MoveL RelTool (p1,64.500000,13.500000,11.989951,\Rx:=0.000000,\Ry:=0.000000),vel1,zoneval,Extruder\WObj:=Workobject_1;
MoveL RelTool (p1,65.000000,13.500000,11.512795,\Rx:=0.000000,\Ry:=0.000000),vel1,zoneval,Extruder\WObj:=Workobject_1;
MoveL RelTool (p1,65.500000,13.500000,11.007442,\Rx:=0.000000,\Ry:=0.000000),vel1,zoneval,Extruder\WObj:=Workobject_1;
MoveL RelTool (p1,66.000000,13.500000,10.423269,\Rx:=0.000000,\Ry:=0.000000),vel1,zoneval,Extruder\WObj:=Workobject_1;
MoveL RelTool (p1,66.500000,13.500000,9.763981,\Rx:=0.000000,\Ry:=0.000000),vel1,zoneval,Extruder\WObj:=Workobject_1;
MoveL RelTool (p1,67.000000,13.500000,9.225973,\Rx:=0.000000,\Ry:=0.000000),vel1,zoneval,Extruder\WObj:=Workobject_1;
MoveL RelTool (p1,67.500000,13.500000,8.874086,\Rx:=0.000000,\Ry:=0.000000),vel1,zoneval,Extruder\WObj:=Workobject_1;
MoveL RelTool (p1,68.000000,13.500000,8.652682,\Rx:=0.000000,\Ry:=0.000000),vel1,zoneval,Extruder\WObj:=Workobject_1;
MoveL RelTool (p1,68.500000,13.500000,8.535785,\Rx:=0.000000,\Ry:=0.000000),vel1,zoneval,Extruder\WObj:=Workobject_1;
MoveL RelTool (p1,69.000000,13.500000,8.500000,\Rx:=0.000000,\Ry:=0.000000),vel1,zoneval,Extruder\WObj:=Workobject_1;
MoveL RelTool (p1,69.500000,13.500000,8.500000,\Rx:=0.000000,\Ry:=0.000000),vel1,zoneval,Extruder\WObj:=Workobject_1;
MoveL RelTool (p1,70.000000,13.500000,8.500000,\Rx:=0.000000,\Ry:=0.000000),vel1,zoneval,Extruder\WObj:=Workobject_1;
MoveL RelTool (p1,70.500000,13.500000,8.500000,\Rx:=0.000000,\Ry:=0.000000),vel1,zoneval,Extruder\WObj:=Workobject_1;
MoveL RelTool (p1,71.000000,13.500000,8.500000,\Rx:=0.000000,\Ry:=0.000000),vel1,zoneval,Extruder\WObj:=Workobject_1;
MoveL RelTool (p1,71.500000,13.500000,8.500000,\Rx:=0.000000,\Ry:=0.000000),vel1,zoneval,Extruder\WObj:=Workobject_1;
MoveL RelTool (p1,72.000000,13.500000,8.500000,\Rx:=0.000000,\Ry:=0.000000),vel1,zoneval,Extruder\WObj:=Workobject_1;
MoveL RelTool (p1,72.500000,13.500000,8.500000,\Rx:=0.000000,\Ry:=0.000000),vel1,zoneval,Extruder\WObj:=Workobject_1;
MoveL RelTool (p1,73.000000,13.500000,8.500000,\Rx:=0.000000,\Ry:=0.000000),vel1,zoneval,Extruder\WObj:=Workobject_1;
MoveL RelTool (p1,73.500000,13.500000,8.500000,\Rx:=0.000000,\Ry:=0.000000),vel1,zoneval,Extruder\WObj:=Workobject_1;
MoveL RelTool (p1,74.000000,13.500000,8.500000,\Rx:=0.000000,\Ry:=0.000000),vel1,zoneval,Extruder\WObj:=Workobject_1;
MoveL RelTool (p1,74.500000,13.500000,8.500000,\Rx:=0.000000,\Ry:=0.000000),vel1,zoneval,Extruder\WObj:=Workobject_1;
MoveL RelTool (p1,75.000000,13.500000,8.500000,\Rx:=0.000000,\Ry:=0.000000),vel1,zoneval,Extruder\WObj:=Workobject_1;
MoveL RelTool (p1,75.500000,13.500000,8.500000,\Rx:=0.000000,\Ry:=0.000000),vel1,zoneval,Extruder\WObj:=Workobject_1;
MoveL RelTool (p1,76.000000,13.500000,8.500000,\Rx:=0.000000,\Ry:=0.000000),vel1,zoneval,Extruder\WObj:=Workobject_1;
MoveL RelTool (p1,76.500000,13.500000,8.500000,\Rx:=0.000000,\Ry:=0.000000),vel1,zoneval,Extruder\WObj:=Workobject_1;
MoveL RelTool (p1,77.000000,13.500000,8.500000,\Rx:=0.000000,\Ry:=0.000000),vel1,zoneval,Extruder\WObj:=Workobject_1;
MoveL RelTool (p1,77.500000,13.500000,8.500000,\Rx:=0.000000,\Ry:=0.000000),vel1,zoneval,Extruder\WObj:=Workobject_1;
MoveL RelTool (p1,78.000000,13.500000,8.500000,\Rx:=0.000000,\Ry:=0.000000),vel1,zoneval,Extruder\WObj:=Workobject_1;
MoveL RelTool (p1,78.500000,13.500000,8.500000,\Rx:=0.000000,\Ry:=0.000000),vel1,zoneval,Extruder\WObj:=Workobject_1;
MoveL RelTool (p1,79.000000,13.500000,8.500000,\Rx:=0.000000,\Ry:=0.000000),vel1,zoneval,Extruder\WObj:=Workobject_1;
MoveL RelTool (p1,79.500000,13.500000,8.500000,\Rx:=0.000000,\Ry:=0.000000),vel1,zoneval,Extruder\WObj:=Workobject_1;
MoveL RelTool (p1,80.000000,13.500000,8.500000,\Rx:=0.000000,\Ry:=0.000000),vel1,zoneval,Extruder\WObj:=Workobject_1;
MoveL RelTool (p1,80.500000,13.500000,8.500000,\Rx:=0.000000,\Ry:=0.000000),vel1,zoneval,Extruder\WObj:=Workobject_1;
MoveL RelTool (p1,81.000000,13.500000,8.500000,\Rx:=0.000000,\Ry:=0.000000),vel1,zoneval,Extruder\WObj:=Workobject_1;
MoveL RelTool (p1,81.500000,13.500000,8.500000,\Rx:=0.000000,\Ry:=0.000000),vel1,zoneval,Extruder\WObj:=Workobject_1;
MoveL RelTool (p1,82.000000,13.500000,8.500000,\Rx:=0.000000,\Ry:=0.000000),vel1,zoneval,Extruder\WObj:=Workobject_1;
MoveL RelTool (p1,82.000000,14.000000,8.500000,\Rx:=0.000000,\Ry:=0.000000),vel1,zoneval,Extruder\WObj:=Workobject_1;
MoveL RelTool (p1,81.500000,14.000000,8.500000,\Rx:=0.000000,\Ry:=0.000000),vel1,zoneval,Extruder\WObj:=Workobject_1;
MoveL RelTool (p1,81.000000,14.000000,8.500000,\Rx:=0.000000,\Ry:=0.000000),vel1,zoneval,Extruder\WObj:=Workobject_1;
MoveL RelTool (p1,80.500000,14.000000,8.500000,\Rx:=0.000000,\Ry:=0.000000),vel1,zoneval,Extruder\WObj:=Workobject_1;
MoveL RelTool (p1,80.000000,14.000000,8.500000,\Rx:=0.000000,\Ry:=0.000000),vel1,zoneval,Extruder\WObj:=Workobject_1;
MoveL RelTool (p1,79.500000,14.000000,8.500000,\Rx:=0.000000,\Ry:=0.000000),vel1,zoneval,Extruder\WObj:=Workobject_1;
MoveL RelTool (p1,79.000000,14.000000,8.500000,\Rx:=0.000000,\Ry:=0.000000),vel1,zoneval,Extruder\WObj:=Workobject_1;
MoveL RelTool (p1,78.500000,14.000000,8.500000,\Rx:=0.000000,\Ry:=0.000000),vel1,zoneval,Extruder\WObj:=Workobject_1;
MoveL RelTool (p1,78.000000,14.000000,8.500000,\Rx:=0.000000,\Ry:=0.000000),vel1,zoneval,Extruder\WObj:=Workobject_1;
MoveL RelTool (p1,77.500000,14.000000,8.500000,\Rx:=0.000000,\Ry:=0.000000),vel1,zoneval,Extruder\WObj:=Workobject_1;
MoveL RelTool (p1,77.000000,14.000000,8.500000,\Rx:=0.000000,\Ry:=0.000000),vel1,zoneval,Extruder\WObj:=Workobject_1;
MoveL RelTool (p1,76.500000,14.000000,8.500000,\Rx:=0.000000,\Ry:=0.000000),vel1,zoneval,Extruder\WObj:=Workobject_1;
MoveL RelTool (p1,76.000000,14.000000,8.500000,\Rx:=0.000000,\Ry:=0.000000),vel1,zoneval,Extruder\WObj:=Workobject_1;
MoveL RelTool (p1,75.500000,14.000000,8.500000,\Rx:=0.000000,\Ry:=0.000000),vel1,zoneval,Extruder\WObj:=Workobject_1;
MoveL RelTool (p1,75.000000,14.000000,8.500000,\Rx:=0.000000,\Ry:=0.000000),vel1,zoneval,Extruder\WObj:=Workobject_1;
MoveL RelTool (p1,74.500000,14.000000,8.500000,\Rx:=0.000000,\Ry:=0.000000),vel1,zoneval,Extruder\WObj:=Workobject_1;
MoveL RelTool (p1,74.000000,14.000000,8.500000,\Rx:=0.000000,\Ry:=0.000000),vel1,zoneval,Extruder\WObj:=Workobject_1;
MoveL RelTool (p1,73.500000,14.000000,8.500000,\Rx:=0.000000,\Ry:=0.000000),vel1,zoneval,Extruder\WObj:=Workobject_1;
MoveL RelTool (p1,73.000000,14.000000,8.500000,\Rx:=0.000000,\Ry:=0.000000),vel1,zoneval,Extruder\WObj:=Workobject_1;
MoveL RelTool (p1,72.500000,14.000000,8.500000,\Rx:=0.000000,\Ry:=0.000000),vel1,zoneval,Extruder\WObj:=Workobject_1;
MoveL RelTool (p1,72.000000,14.000000,8.500000,\Rx:=0.000000,\Ry:=0.000000),vel1,zoneval,Extruder\WObj:=Workobject_1;
MoveL RelTool (p1,71.500000,14.000000,8.500000,\Rx:=0.000000,\Ry:=0.000000),vel1,zoneval,Extruder\WObj:=Workobject_1;
MoveL RelTool (p1,71.000000,14.000000,8.500000,\Rx:=0.000000,\Ry:=0.000000),vel1,zoneval,Extruder\WObj:=Workobject_1;
MoveL RelTool (p1,70.500000,14.000000,8.500000,\Rx:=0.000000,\Ry:=0.000000),vel1,zoneval,Extruder\WObj:=Workobject_1;
MoveL RelTool (p1,70.000000,14.000000,8.500000,\Rx:=0.000000,\Ry:=0.000000),vel1,zoneval,Extruder\WObj:=Workobject_1;
MoveL RelTool (p1,69.500000,14.000000,8.500000,\Rx:=0.000000,\Ry:=0.000000),vel1,zoneval,Extruder\WObj:=Workobject_1;
MoveL RelTool (p1,69.000000,14.000000,8.500000,\Rx:=0.000000,\Ry:=0.000000),vel1,zoneval,Extruder\WObj:=Workobject_1;
MoveL RelTool (p1,68.500000,14.000000,8.535785,\Rx:=0.000000,\Ry:=0.000000),vel1,zoneval,Extruder\WObj:=Workobject_1;
MoveL RelTool (p1,68.000000,14.000000,8.652682,\Rx:=0.000000,\Ry:=0.000000),vel1,zoneval,Extruder\WObj:=Workobject_1;
MoveL RelTool (p1,67.500000,14.000000,8.874086,\Rx:=0.000000,\Ry:=0.000000),vel1,zoneval,Extruder\WObj:=Workobject_1;
MoveL RelTool (p1,67.000000,14.000000,9.225973,\Rx:=0.000000,\Ry:=0.000000),vel1,zoneval,Extruder\WObj:=Workobject_1;
MoveL RelTool (p1,66.500000,14.000000,9.763981,\Rx:=0.000000,\Ry:=0.000000),vel1,zoneval,Extruder\WObj:=Workobject_1;
MoveL RelTool (p1,66.000000,14.000000,10.424782,\Rx:=0.000000,\Ry:=0.000000),vel1,zoneval,Extruder\WObj:=Workobject_1;
MoveL RelTool (p1,65.500000,14.000000,11.007081,\Rx:=0.000000,\Ry:=0.000000),vel1,zoneval,Extruder\WObj:=Workobject_1;
MoveL RelTool (p1,65.000000,14.000000,11.513962,\Rx:=0.000000,\Ry:=0.000000),vel1,zoneval,Extruder\WObj:=Workobject_1;
MoveL RelTool (p1,64.500000,14.000000,11.989543,\Rx:=0.000000,\Ry:=0.000000),vel1,zoneval,Extruder\WObj:=Workobject_1;
MoveL RelTool (p1,64.000000,14.000000,12.421528,\Rx:=0.000000,\Ry:=0.000000),vel1,zoneval,Extruder\WObj:=Workobject_1;
MoveL RelTool (p1,63.500000,14.000000,12.805855,\Rx:=0.000000,\Ry:=0.000000),vel1,zoneval,Extruder\WObj:=Workobject_1;
MoveL RelTool (p1,63.000000,14.000000,13.179500,\Rx:=0.000000,\Ry:=0.000000),vel1,zoneval,Extruder\WObj:=Workobject_1;
MoveL RelTool (p1,62.500000,14.000000,13.514872,\Rx:=0.000000,\Ry:=0.000000),vel1,zoneval,Extruder\WObj:=Workobject_1;
MoveL RelTool (p1,62.000000,14.000000,13.838447,\Rx:=0.000000,\Ry:=0.000000),vel1,zoneval,Extruder\WObj:=Workobject_1;
MoveL RelTool (p1,61.500000,14.000000,14.134422,\Rx:=0.000000,\Ry:=0.000000),vel1,zoneval,Extruder\WObj:=Workobject_1;
MoveL RelTool (p1,61.000000,14.000000,14.418567,\Rx:=0.000000,\Ry:=0.000000),vel1,zoneval,Extruder\WObj:=Workobject_1;
MoveL RelTool (p1,60.500000,14.000000,14.677184,\Rx:=0.000000,\Ry:=0.000000),vel1,zoneval,Extruder\WObj:=Workobject_1;
MoveL RelTool (p1,60.000000,14.000000,14.938229,\Rx:=0.000000,\Ry:=0.000000),vel1,zoneval,Extruder\WObj:=Workobject_1;
MoveL RelTool (p1,59.500000,14.000000,15.174609,\Rx:=0.000000,\Ry:=0.000000),vel1,zoneval,Extruder\WObj:=Workobject_1;
MoveL RelTool (p1,59.000000,14.000000,15.404406,\Rx:=0.000000,\Ry:=0.000000),vel1,zoneval,Extruder\WObj:=Workobject_1;
MoveL RelTool (p1,58.500000,14.000000,15.614404,\Rx:=0.000000,\Ry:=0.000000),vel1,zoneval,Extruder\WObj:=Workobject_1;
MoveL RelTool (p1,58.000000,14.000000,15.816030,\Rx:=0.000000,\Ry:=0.000000),vel1,zoneval,Extruder\WObj:=Workobject_1;
MoveL RelTool (p1,57.500000,14.000000,16.017656,\Rx:=0.000000,\Ry:=0.000000),vel1,zoneval,Extruder\WObj:=Workobject_1;
MoveL RelTool (p1,57.000000,14.000000,16.197291,\Rx:=0.000000,\Ry:=0.000000),vel1,zoneval,Extruder\WObj:=Workobject_1;
MoveL RelTool (p1,56.500000,14.000000,16.373201,\Rx:=0.000000,\Ry:=0.000000),vel1,zoneval,Extruder\WObj:=Workobject_1;
MoveL RelTool (p1,56.000000,14.000000,16.541775,\Rx:=0.000000,\Ry:=0.000000),vel1,zoneval,Extruder\WObj:=Workobject_1;
MoveL RelTool (p1,55.500000,14.000000,16.695933,\Rx:=0.000000,\Ry:=0.000000),vel1,zoneval,Extruder\WObj:=Workobject_1;
MoveL RelTool (p1,55.000000,14.000000,16.847549,\Rx:=0.000000,\Ry:=0.000000),vel1,zoneval,Extruder\WObj:=Workobject_1;
MoveL RelTool (p1,54.500000,14.000000,16.992424,\Rx:=0.000000,\Ry:=0.000000),vel1,zoneval,Extruder\WObj:=Workobject_1;
MoveL RelTool (p1,54.000000,14.000000,17.116147,\Rx:=0.000000,\Ry:=0.000000),vel1,zoneval,Extruder\WObj:=Workobject_1;
MoveL RelTool (p1,53.500000,14.000000,17.244747,\Rx:=0.000000,\Ry:=0.000000),vel1,zoneval,Extruder\WObj:=Workobject_1;
MoveL RelTool (p1,53.000000,14.000000,17.373347,\Rx:=0.000000,\Ry:=0.000000),vel1,zoneval,Extruder\WObj:=Workobject_1;
MoveL RelTool (p1,52.500000,14.000000,17.484402,\Rx:=0.000000,\Ry:=0.000000),vel1,zoneval,Extruder\WObj:=Workobject_1;
MoveL RelTool (p1,52.000000,14.000000,17.591158,\Rx:=0.000000,\Ry:=0.000000),vel1,zoneval,Extruder\WObj:=Workobject_1;
MoveL RelTool (p1,51.500000,14.000000,17.695333,\Rx:=0.000000,\Ry:=0.000000),vel1,zoneval,Extruder\WObj:=Workobject_1;
MoveL RelTool (p1,51.000000,14.000000,17.779951,\Rx:=0.000000,\Ry:=0.000000),vel1,zoneval,Extruder\WObj:=Workobject_1;
MoveL RelTool (p1,50.500000,14.000000,17.865927,\Rx:=0.000000,\Ry:=0.000000),vel1,zoneval,Extruder\WObj:=Workobject_1;
MoveL RelTool (p1,50.000000,14.000000,17.951904,\Rx:=0.000000,\Ry:=0.000000),vel1,zoneval,Extruder\WObj:=Workobject_1;
MoveL RelTool (p1,49.500000,14.000000,18.029069,\Rx:=0.000000,\Ry:=0.000000),vel1,zoneval,Extruder\WObj:=Workobject_1;
MoveL RelTool (p1,49.000000,14.000000,18.095126,\Rx:=0.000000,\Ry:=0.000000),vel1,zoneval,Extruder\WObj:=Workobject_1;
MoveL RelTool (p1,48.500000,14.000000,18.161183,\Rx:=0.000000,\Ry:=0.000000),vel1,zoneval,Extruder\WObj:=Workobject_1;
MoveL RelTool (p1,48.000000,14.000000,18.218591,\Rx:=0.000000,\Ry:=0.000000),vel1,zoneval,Extruder\WObj:=Workobject_1;
MoveL RelTool (p1,47.500000,14.000000,18.266605,\Rx:=0.000000,\Ry:=0.000000),vel1,zoneval,Extruder\WObj:=Workobject_1;
MoveL RelTool (p1,47.000000,14.000000,18.313237,\Rx:=0.000000,\Ry:=0.000000),vel1,zoneval,Extruder\WObj:=Workobject_1;
MoveL RelTool (p1,46.500000,14.000000,18.359868,\Rx:=0.000000,\Ry:=0.000000),vel1,zoneval,Extruder\WObj:=Workobject_1;
MoveL RelTool (p1,46.000000,14.000000,18.393525,\Rx:=0.000000,\Ry:=0.000000),vel1,zoneval,Extruder\WObj:=Workobject_1;
MoveL RelTool (p1,45.500000,14.000000,18.421069,\Rx:=0.000000,\Ry:=0.000000),vel1,zoneval,Extruder\WObj:=Workobject_1;
MoveL RelTool (p1,45.000000,14.000000,18.448613,\Rx:=0.000000,\Ry:=0.000000),vel1,zoneval,Extruder\WObj:=Workobject_1;
MoveL RelTool (p1,44.500000,14.000000,18.469450,\Rx:=0.000000,\Ry:=0.000000),vel1,zoneval,Extruder\WObj:=Workobject_1;
MoveL RelTool (p1,44.000000,14.000000,18.480446,\Rx:=0.000000,\Ry:=0.000000),vel1,zoneval,Extruder\WObj:=Workobject_1;
MoveL RelTool (p1,43.500000,14.000000,18.488975,\Rx:=0.000000,\Ry:=0.000000),vel1,zoneval,Extruder\WObj:=Workobject_1;
MoveL RelTool (p1,43.000000,14.000000,18.497504,\Rx:=0.000000,\Ry:=0.000000),vel1,zoneval,Extruder\WObj:=Workobject_1;
MoveL RelTool (p1,42.500000,14.000000,18.493713,\Rx:=0.000000,\Ry:=0.000000),vel1,zoneval,Extruder\WObj:=Workobject_1;
MoveL RelTool (p1,42.000000,14.000000,18.483301,\Rx:=0.000000,\Ry:=0.000000),vel1,zoneval,Extruder\WObj:=Workobject_1;
MoveL RelTool (p1,41.500000,14.000000,18.472889,\Rx:=0.000000,\Ry:=0.000000),vel1,zoneval,Extruder\WObj:=Workobject_1;
MoveL RelTool (p1,41.000000,14.000000,18.457063,\Rx:=0.000000,\Ry:=0.000000),vel1,zoneval,Extruder\WObj:=Workobject_1;
MoveL RelTool (p1,40.500000,14.000000,18.431185,\Rx:=0.000000,\Ry:=0.000000),vel1,zoneval,Extruder\WObj:=Workobject_1;
MoveL RelTool (p1,40.000000,14.000000,18.401735,\Rx:=0.000000,\Ry:=0.000000),vel1,zoneval,Extruder\WObj:=Workobject_1;
MoveL RelTool (p1,39.500000,14.000000,18.372284,\Rx:=0.000000,\Ry:=0.000000),vel1,zoneval,Extruder\WObj:=Workobject_1;
MoveL RelTool (p1,39.000000,14.000000,18.328181,\Rx:=0.000000,\Ry:=0.000000),vel1,zoneval,Extruder\WObj:=Workobject_1;
MoveL RelTool (p1,38.500000,14.000000,18.278194,\Rx:=0.000000,\Ry:=0.000000),vel1,zoneval,Extruder\WObj:=Workobject_1;
MoveL RelTool (p1,38.000000,14.000000,18.229591,\Rx:=0.000000,\Ry:=0.000000),vel1,zoneval,Extruder\WObj:=Workobject_1;
MoveL RelTool (p1,37.500000,14.000000,18.180988,\Rx:=0.000000,\Ry:=0.000000),vel1,zoneval,Extruder\WObj:=Workobject_1;
MoveL RelTool (p1,37.000000,14.000000,18.118155,\Rx:=0.000000,\Ry:=0.000000),vel1,zoneval,Extruder\WObj:=Workobject_1;
MoveL RelTool (p1,36.500000,14.000000,18.049890,\Rx:=0.000000,\Ry:=0.000000),vel1,zoneval,Extruder\WObj:=Workobject_1;
MoveL RelTool (p1,36.000000,14.000000,17.981627,\Rx:=0.000000,\Ry:=0.000000),vel1,zoneval,Extruder\WObj:=Workobject_1;
MoveL RelTool (p1,35.500000,14.000000,17.897001,\Rx:=0.000000,\Ry:=0.000000),vel1,zoneval,Extruder\WObj:=Workobject_1;
MoveL RelTool (p1,35.000000,14.000000,17.808427,\Rx:=0.000000,\Ry:=0.000000),vel1,zoneval,Extruder\WObj:=Workobject_1;
MoveL RelTool (p1,34.500000,14.000000,17.719854,\Rx:=0.000000,\Ry:=0.000000),vel1,zoneval,Extruder\WObj:=Workobject_1;
MoveL RelTool (p1,34.000000,14.000000,17.630421,\Rx:=0.000000,\Ry:=0.000000),vel1,zoneval,Extruder\WObj:=Workobject_1;
MoveL RelTool (p1,33.500000,14.000000,17.520494,\Rx:=0.000000,\Ry:=0.000000),vel1,zoneval,Extruder\WObj:=Workobject_1;
MoveL RelTool (p1,33.000000,14.000000,17.410567,\Rx:=0.000000,\Ry:=0.000000),vel1,zoneval,Extruder\WObj:=Workobject_1;
MoveL RelTool (p1,32.500000,14.000000,17.295270,\Rx:=0.000000,\Ry:=0.000000),vel1,zoneval,Extruder\WObj:=Workobject_1;
MoveL RelTool (p1,32.000000,14.000000,17.166180,\Rx:=0.000000,\Ry:=0.000000),vel1,zoneval,Extruder\WObj:=Workobject_1;
MoveL RelTool (p1,31.500000,14.000000,17.033775,\Rx:=0.000000,\Ry:=0.000000),vel1,zoneval,Extruder\WObj:=Workobject_1;
MoveL RelTool (p1,31.000000,14.000000,16.901371,\Rx:=0.000000,\Ry:=0.000000),vel1,zoneval,Extruder\WObj:=Workobject_1;
MoveL RelTool (p1,30.500000,14.000000,16.748138,\Rx:=0.000000,\Ry:=0.000000),vel1,zoneval,Extruder\WObj:=Workobject_1;
MoveL RelTool (p1,30.000000,14.000000,16.592069,\Rx:=0.000000,\Ry:=0.000000),vel1,zoneval,Extruder\WObj:=Workobject_1;
MoveL RelTool (p1,29.500000,14.000000,16.432055,\Rx:=0.000000,\Ry:=0.000000),vel1,zoneval,Extruder\WObj:=Workobject_1;
MoveL RelTool (p1,29.000000,14.000000,16.256775,\Rx:=0.000000,\Ry:=0.000000),vel1,zoneval,Extruder\WObj:=Workobject_1;
MoveL RelTool (p1,28.500000,14.000000,16.075776,\Rx:=0.000000,\Ry:=0.000000),vel1,zoneval,Extruder\WObj:=Workobject_1;
MoveL RelTool (p1,28.000000,14.000000,15.889441,\Rx:=0.000000,\Ry:=0.000000),vel1,zoneval,Extruder\WObj:=Workobject_1;
MoveL RelTool (p1,27.500000,14.000000,15.681605,\Rx:=0.000000,\Ry:=0.000000),vel1,zoneval,Extruder\WObj:=Workobject_1;
MoveL RelTool (p1,27.000000,14.000000,15.473770,\Rx:=0.000000,\Ry:=0.000000),vel1,zoneval,Extruder\WObj:=Workobject_1;
MoveL RelTool (p1,26.500000,14.000000,15.254742,\Rx:=0.000000,\Ry:=0.000000),vel1,zoneval,Extruder\WObj:=Workobject_1;
MoveL RelTool (p1,26.000000,14.000000,15.016990,\Rx:=0.000000,\Ry:=0.000000),vel1,zoneval,Extruder\WObj:=Workobject_1;
MoveL RelTool (p1,25.500000,14.000000,14.773856,\Rx:=0.000000,\Ry:=0.000000),vel1,zoneval,Extruder\WObj:=Workobject_1;
MoveL RelTool (p1,25.000000,14.000000,14.503734,\Rx:=0.000000,\Ry:=0.000000),vel1,zoneval,Extruder\WObj:=Workobject_1;
MoveL RelTool (p1,24.500000,14.000000,14.232533,\Rx:=0.000000,\Ry:=0.000000),vel1,zoneval,Extruder\WObj:=Workobject_1;
MoveL RelTool (p1,24.000000,14.000000,13.937132,\Rx:=0.000000,\Ry:=0.000000),vel1,zoneval,Extruder\WObj:=Workobject_1;
MoveL RelTool (p1,23.500000,14.000000,13.628434,\Rx:=0.000000,\Ry:=0.000000),vel1,zoneval,Extruder\WObj:=Workobject_1;
MoveL RelTool (p1,23.000000,14.000000,13.289112,\Rx:=0.000000,\Ry:=0.000000),vel1,zoneval,Extruder\WObj:=Workobject_1;
MoveL RelTool (p1,22.500000,14.000000,12.938180,\Rx:=0.000000,\Ry:=0.000000),vel1,zoneval,Extruder\WObj:=Workobject_1;
MoveL RelTool (p1,22.000000,14.000000,12.548317,\Rx:=0.000000,\Ry:=0.000000),vel1,zoneval,Extruder\WObj:=Workobject_1;
MoveL RelTool (p1,21.500000,14.000000,12.139462,\Rx:=0.000000,\Ry:=0.000000),vel1,zoneval,Extruder\WObj:=Workobject_1;
MoveL RelTool (p1,21.000000,14.000000,11.683424,\Rx:=0.000000,\Ry:=0.000000),vel1,zoneval,Extruder\WObj:=Workobject_1;
MoveL RelTool (p1,20.500000,14.000000,11.178595,\Rx:=0.000000,\Ry:=0.000000),vel1,zoneval,Extruder\WObj:=Workobject_1;
MoveL RelTool (p1,20.000000,14.000000,10.625965,\Rx:=0.000000,\Ry:=0.000000),vel1,zoneval,Extruder\WObj:=Workobject_1;
MoveL RelTool (p1,19.500000,14.000000,9.992651,\Rx:=0.000000,\Ry:=0.000000),vel1,zoneval,Extruder\WObj:=Workobject_1;
MoveL RelTool (p1,19.000000,14.000000,9.374813,\Rx:=0.000000,\Ry:=0.000000),vel1,zoneval,Extruder\WObj:=Workobject_1;
MoveL RelTool (p1,18.500000,14.000000,8.980296,\Rx:=0.000000,\Ry:=0.000000),vel1,zoneval,Extruder\WObj:=Workobject_1;
MoveL RelTool (p1,18.000000,14.000000,8.722633,\Rx:=0.000000,\Ry:=0.000000),vel1,zoneval,Extruder\WObj:=Workobject_1;
MoveL RelTool (p1,17.500000,14.000000,8.570628,\Rx:=0.000000,\Ry:=0.000000),vel1,zoneval,Extruder\WObj:=Workobject_1;
MoveL RelTool (p1,17.000000,14.000000,8.508911,\Rx:=0.000000,\Ry:=0.000000),vel1,zoneval,Extruder\WObj:=Workobject_1;
MoveL RelTool (p1,16.500000,14.000000,8.500000,\Rx:=0.000000,\Ry:=0.000000),vel1,zoneval,Extruder\WObj:=Workobject_1;
MoveL RelTool (p1,16.000000,14.000000,8.500000,\Rx:=0.000000,\Ry:=0.000000),vel1,zoneval,Extruder\WObj:=Workobject_1;
MoveL RelTool (p1,15.500000,14.000000,8.500000,\Rx:=0.000000,\Ry:=0.000000),vel1,zoneval,Extruder\WObj:=Workobject_1;
MoveL RelTool (p1,15.000000,14.000000,8.500000,\Rx:=0.000000,\Ry:=0.000000),vel1,zoneval,Extruder\WObj:=Workobject_1;
MoveL RelTool (p1,14.500000,14.000000,8.500000,\Rx:=0.000000,\Ry:=0.000000),vel1,zoneval,Extruder\WObj:=Workobject_1;
MoveL RelTool (p1,14.000000,14.000000,8.500000,\Rx:=0.000000,\Ry:=0.000000),vel1,zoneval,Extruder\WObj:=Workobject_1;
MoveL RelTool (p1,13.500000,14.000000,8.500000,\Rx:=0.000000,\Ry:=0.000000),vel1,zoneval,Extruder\WObj:=Workobject_1;
MoveL RelTool (p1,13.000000,14.000000,8.500000,\Rx:=0.000000,\Ry:=0.000000),vel1,zoneval,Extruder\WObj:=Workobject_1;
MoveL RelTool (p1,12.500000,14.000000,8.500000,\Rx:=0.000000,\Ry:=0.000000),vel1,zoneval,Extruder\WObj:=Workobject_1;
MoveL RelTool (p1,12.000000,14.000000,8.500000,\Rx:=0.000000,\Ry:=0.000000),vel1,zoneval,Extruder\WObj:=Workobject_1;
MoveL RelTool (p1,11.500000,14.000000,8.500000,\Rx:=0.000000,\Ry:=0.000000),vel1,zoneval,Extruder\WObj:=Workobject_1;
MoveL RelTool (p1,11.000000,14.000000,8.500000,\Rx:=0.000000,\Ry:=0.000000),vel1,zoneval,Extruder\WObj:=Workobject_1;
MoveL RelTool (p1,10.500000,14.000000,8.500000,\Rx:=0.000000,\Ry:=0.000000),vel1,zoneval,Extruder\WObj:=Workobject_1;
MoveL RelTool (p1,10.000000,14.000000,8.500000,\Rx:=0.000000,\Ry:=0.000000),vel1,zoneval,Extruder\WObj:=Workobject_1;
MoveL RelTool (p1,9.500000,14.000000,8.500000,\Rx:=0.000000,\Ry:=0.000000),vel1,zoneval,Extruder\WObj:=Workobject_1;
MoveL RelTool (p1,9.000000,14.000000,8.500000,\Rx:=0.000000,\Ry:=0.000000),vel1,zoneval,Extruder\WObj:=Workobject_1;
MoveL RelTool (p1,8.500000,14.000000,8.500000,\Rx:=0.000000,\Ry:=0.000000),vel1,zoneval,Extruder\WObj:=Workobject_1;
MoveL RelTool (p1,8.000000,14.000000,8.500000,\Rx:=0.000000,\Ry:=0.000000),vel1,zoneval,Extruder\WObj:=Workobject_1;
MoveL RelTool (p1,7.500000,14.000000,8.500000,\Rx:=0.000000,\Ry:=0.000000),vel1,zoneval,Extruder\WObj:=Workobject_1;
MoveL RelTool (p1,7.000000,14.000000,8.500000,\Rx:=0.000000,\Ry:=0.000000),vel1,zoneval,Extruder\WObj:=Workobject_1;
MoveL RelTool (p1,6.500000,14.000000,8.500000,\Rx:=0.000000,\Ry:=0.000000),vel1,zoneval,Extruder\WObj:=Workobject_1;
MoveL RelTool (p1,6.000000,14.000000,8.500000,\Rx:=0.000000,\Ry:=0.000000),vel1,zoneval,Extruder\WObj:=Workobject_1;
MoveL RelTool (p1,5.500000,14.000000,8.500000,\Rx:=0.000000,\Ry:=0.000000),vel1,zoneval,Extruder\WObj:=Workobject_1;
MoveL RelTool (p1,5.000000,14.000000,8.500000,\Rx:=0.000000,\Ry:=0.000000),vel1,zoneval,Extruder\WObj:=Workobject_1;
MoveL RelTool (p1,4.500000,14.000000,8.500000,\Rx:=0.000000,\Ry:=0.000000),vel1,zoneval,Extruder\WObj:=Workobject_1;
MoveL RelTool (p1,4.000000,14.000000,8.500000,\Rx:=0.000000,\Ry:=0.000000),vel1,zoneval,Extruder\WObj:=Workobject_1;
MoveL RelTool (p1,3.500000,14.000000,8.500000,\Rx:=0.000000,\Ry:=0.000000),vel1,zoneval,Extruder\WObj:=Workobject_1;
MoveL RelTool (p1,3.500000,14.500000,8.500000,\Rx:=0.000000,\Ry:=0.000000),vel1,zoneval,Extruder\WObj:=Workobject_1;
MoveL RelTool (p1,4.000000,14.500000,8.500000,\Rx:=0.000000,\Ry:=0.000000),vel1,zoneval,Extruder\WObj:=Workobject_1;
MoveL RelTool (p1,4.500000,14.500000,8.500000,\Rx:=0.000000,\Ry:=0.000000),vel1,zoneval,Extruder\WObj:=Workobject_1;
MoveL RelTool (p1,5.000000,14.500000,8.500000,\Rx:=0.000000,\Ry:=0.000000),vel1,zoneval,Extruder\WObj:=Workobject_1;
MoveL RelTool (p1,5.500000,14.500000,8.500000,\Rx:=0.000000,\Ry:=0.000000),vel1,zoneval,Extruder\WObj:=Workobject_1;
MoveL RelTool (p1,6.000000,14.500000,8.500000,\Rx:=0.000000,\Ry:=0.000000),vel1,zoneval,Extruder\WObj:=Workobject_1;
MoveL RelTool (p1,6.500000,14.500000,8.500000,\Rx:=0.000000,\Ry:=0.000000),vel1,zoneval,Extruder\WObj:=Workobject_1;
MoveL RelTool (p1,7.000000,14.500000,8.500000,\Rx:=0.000000,\Ry:=0.000000),vel1,zoneval,Extruder\WObj:=Workobject_1;
MoveL RelTool (p1,7.500000,14.500000,8.500000,\Rx:=0.000000,\Ry:=0.000000),vel1,zoneval,Extruder\WObj:=Workobject_1;
MoveL RelTool (p1,8.000000,14.500000,8.500000,\Rx:=0.000000,\Ry:=0.000000),vel1,zoneval,Extruder\WObj:=Workobject_1;
MoveL RelTool (p1,8.500000,14.500000,8.500000,\Rx:=0.000000,\Ry:=0.000000),vel1,zoneval,Extruder\WObj:=Workobject_1;
MoveL RelTool (p1,9.000000,14.500000,8.500000,\Rx:=0.000000,\Ry:=0.000000),vel1,zoneval,Extruder\WObj:=Workobject_1;
MoveL RelTool (p1,9.500000,14.500000,8.500000,\Rx:=0.000000,\Ry:=0.000000),vel1,zoneval,Extruder\WObj:=Workobject_1;
MoveL RelTool (p1,10.000000,14.500000,8.500000,\Rx:=0.000000,\Ry:=0.000000),vel1,zoneval,Extruder\WObj:=Workobject_1;
MoveL RelTool (p1,10.500000,14.500000,8.500000,\Rx:=0.000000,\Ry:=0.000000),vel1,zoneval,Extruder\WObj:=Workobject_1;
MoveL RelTool (p1,11.000000,14.500000,8.500000,\Rx:=0.000000,\Ry:=0.000000),vel1,zoneval,Extruder\WObj:=Workobject_1;
MoveL RelTool (p1,11.500000,14.500000,8.500000,\Rx:=0.000000,\Ry:=0.000000),vel1,zoneval,Extruder\WObj:=Workobject_1;
MoveL RelTool (p1,12.000000,14.500000,8.500000,\Rx:=0.000000,\Ry:=0.000000),vel1,zoneval,Extruder\WObj:=Workobject_1;
MoveL RelTool (p1,12.500000,14.500000,8.500000,\Rx:=0.000000,\Ry:=0.000000),vel1,zoneval,Extruder\WObj:=Workobject_1;
MoveL RelTool (p1,13.000000,14.500000,8.500000,\Rx:=0.000000,\Ry:=0.000000),vel1,zoneval,Extruder\WObj:=Workobject_1;
MoveL RelTool (p1,13.500000,14.500000,8.500000,\Rx:=0.000000,\Ry:=0.000000),vel1,zoneval,Extruder\WObj:=Workobject_1;
MoveL RelTool (p1,14.000000,14.500000,8.500000,\Rx:=0.000000,\Ry:=0.000000),vel1,zoneval,Extruder\WObj:=Workobject_1;
MoveL RelTool (p1,14.500000,14.500000,8.500000,\Rx:=0.000000,\Ry:=0.000000),vel1,zoneval,Extruder\WObj:=Workobject_1;
MoveL RelTool (p1,15.000000,14.500000,8.500000,\Rx:=0.000000,\Ry:=0.000000),vel1,zoneval,Extruder\WObj:=Workobject_1;
MoveL RelTool (p1,15.500000,14.500000,8.500000,\Rx:=0.000000,\Ry:=0.000000),vel1,zoneval,Extruder\WObj:=Workobject_1;
MoveL RelTool (p1,16.000000,14.500000,8.500000,\Rx:=0.000000,\Ry:=0.000000),vel1,zoneval,Extruder\WObj:=Workobject_1;
MoveL RelTool (p1,16.500000,14.500000,8.500000,\Rx:=0.000000,\Ry:=0.000000),vel1,zoneval,Extruder\WObj:=Workobject_1;
MoveL RelTool (p1,17.000000,14.500000,8.508911,\Rx:=0.000000,\Ry:=0.000000),vel1,zoneval,Extruder\WObj:=Workobject_1;
MoveL RelTool (p1,17.500000,14.500000,8.570628,\Rx:=0.000000,\Ry:=0.000000),vel1,zoneval,Extruder\WObj:=Workobject_1;
MoveL RelTool (p1,18.000000,14.500000,8.722633,\Rx:=0.000000,\Ry:=0.000000),vel1,zoneval,Extruder\WObj:=Workobject_1;
MoveL RelTool (p1,18.500000,14.500000,8.980296,\Rx:=0.000000,\Ry:=0.000000),vel1,zoneval,Extruder\WObj:=Workobject_1;
MoveL RelTool (p1,19.000000,14.500000,9.374813,\Rx:=0.000000,\Ry:=0.000000),vel1,zoneval,Extruder\WObj:=Workobject_1;
MoveL RelTool (p1,19.500000,14.500000,9.992651,\Rx:=0.000000,\Ry:=0.000000),vel1,zoneval,Extruder\WObj:=Workobject_1;
MoveL RelTool (p1,20.000000,14.500000,10.625441,\Rx:=0.000000,\Ry:=0.000000),vel1,zoneval,Extruder\WObj:=Workobject_1;
MoveL RelTool (p1,20.500000,14.500000,11.179034,\Rx:=0.000000,\Ry:=0.000000),vel1,zoneval,Extruder\WObj:=Workobject_1;
MoveL RelTool (p1,21.000000,14.500000,11.683147,\Rx:=0.000000,\Ry:=0.000000),vel1,zoneval,Extruder\WObj:=Workobject_1;
MoveL RelTool (p1,21.500000,14.500000,12.140800,\Rx:=0.000000,\Ry:=0.000000),vel1,zoneval,Extruder\WObj:=Workobject_1;
MoveL RelTool (p1,22.000000,14.500000,12.548217,\Rx:=0.000000,\Ry:=0.000000),vel1,zoneval,Extruder\WObj:=Workobject_1;
MoveL RelTool (p1,22.500000,14.500000,12.938300,\Rx:=0.000000,\Ry:=0.000000),vel1,zoneval,Extruder\WObj:=Workobject_1;
MoveL RelTool (p1,23.000000,14.500000,13.289231,\Rx:=0.000000,\Ry:=0.000000),vel1,zoneval,Extruder\WObj:=Workobject_1;
MoveL RelTool (p1,23.500000,14.500000,13.628094,\Rx:=0.000000,\Ry:=0.000000),vel1,zoneval,Extruder\WObj:=Workobject_1;
MoveL RelTool (p1,24.000000,14.500000,13.936792,\Rx:=0.000000,\Ry:=0.000000),vel1,zoneval,Extruder\WObj:=Workobject_1;
MoveL RelTool (p1,24.500000,14.500000,14.233179,\Rx:=0.000000,\Ry:=0.000000),vel1,zoneval,Extruder\WObj:=Workobject_1;
MoveL RelTool (p1,25.000000,14.500000,14.504380,\Rx:=0.000000,\Ry:=0.000000),vel1,zoneval,Extruder\WObj:=Workobject_1;
MoveL RelTool (p1,25.500000,14.500000,14.774776,\Rx:=0.000000,\Ry:=0.000000),vel1,zoneval,Extruder\WObj:=Workobject_1;
MoveL RelTool (p1,26.000000,14.500000,15.016632,\Rx:=0.000000,\Ry:=0.000000),vel1,zoneval,Extruder\WObj:=Workobject_1;
MoveL RelTool (p1,26.500000,14.500000,15.254383,\Rx:=0.000000,\Ry:=0.000000),vel1,zoneval,Extruder\WObj:=Workobject_1;
MoveL RelTool (p1,27.000000,14.500000,15.474110,\Rx:=0.000000,\Ry:=0.000000),vel1,zoneval,Extruder\WObj:=Workobject_1;
MoveL RelTool (p1,27.500000,14.500000,15.681946,\Rx:=0.000000,\Ry:=0.000000),vel1,zoneval,Extruder\WObj:=Workobject_1;
MoveL RelTool (p1,28.000000,14.500000,15.889782,\Rx:=0.000000,\Ry:=0.000000),vel1,zoneval,Extruder\WObj:=Workobject_1;
MoveL RelTool (p1,28.500000,14.500000,16.075557,\Rx:=0.000000,\Ry:=0.000000),vel1,zoneval,Extruder\WObj:=Workobject_1;
MoveL RelTool (p1,29.000000,14.500000,16.256557,\Rx:=0.000000,\Ry:=0.000000),vel1,zoneval,Extruder\WObj:=Workobject_1;
MoveL RelTool (p1,29.500000,14.500000,16.433092,\Rx:=0.000000,\Ry:=0.000000),vel1,zoneval,Extruder\WObj:=Workobject_1;
MoveL RelTool (p1,30.000000,14.500000,16.591990,\Rx:=0.000000,\Ry:=0.000000),vel1,zoneval,Extruder\WObj:=Workobject_1;
MoveL RelTool (p1,30.500000,14.500000,16.748059,\Rx:=0.000000,\Ry:=0.000000),vel1,zoneval,Extruder\WObj:=Workobject_1;
MoveL RelTool (p1,31.000000,14.500000,16.901521,\Rx:=0.000000,\Ry:=0.000000),vel1,zoneval,Extruder\WObj:=Workobject_1;
MoveL RelTool (p1,31.500000,14.500000,17.033926,\Rx:=0.000000,\Ry:=0.000000),vel1,zoneval,Extruder\WObj:=Workobject_1;
MoveL RelTool (p1,32.000000,14.500000,17.166330,\Rx:=0.000000,\Ry:=0.000000),vel1,zoneval,Extruder\WObj:=Workobject_1;
MoveL RelTool (p1,32.500000,14.500000,17.296270,\Rx:=0.000000,\Ry:=0.000000),vel1,zoneval,Extruder\WObj:=Workobject_1;
MoveL RelTool (p1,33.000000,14.500000,17.410275,\Rx:=0.000000,\Ry:=0.000000),vel1,zoneval,Extruder\WObj:=Workobject_1;
MoveL RelTool (p1,33.500000,14.500000,17.520202,\Rx:=0.000000,\Ry:=0.000000),vel1,zoneval,Extruder\WObj:=Workobject_1;
MoveL RelTool (p1,34.000000,14.500000,17.630129,\Rx:=0.000000,\Ry:=0.000000),vel1,zoneval,Extruder\WObj:=Workobject_1;
MoveL RelTool (p1,34.500000,14.500000,17.720622,\Rx:=0.000000,\Ry:=0.000000),vel1,zoneval,Extruder\WObj:=Workobject_1;
MoveL RelTool (p1,35.000000,14.500000,17.809195,\Rx:=0.000000,\Ry:=0.000000),vel1,zoneval,Extruder\WObj:=Workobject_1;
MoveL RelTool (p1,35.500000,14.500000,17.897769,\Rx:=0.000000,\Ry:=0.000000),vel1,zoneval,Extruder\WObj:=Workobject_1;
MoveL RelTool (p1,36.000000,14.500000,17.981309,\Rx:=0.000000,\Ry:=0.000000),vel1,zoneval,Extruder\WObj:=Workobject_1;
MoveL RelTool (p1,36.500000,14.500000,18.049573,\Rx:=0.000000,\Ry:=0.000000),vel1,zoneval,Extruder\WObj:=Workobject_1;
MoveL RelTool (p1,37.000000,14.500000,18.117838,\Rx:=0.000000,\Ry:=0.000000),vel1,zoneval,Extruder\WObj:=Workobject_1;
MoveL RelTool (p1,37.500000,14.500000,18.182228,\Rx:=0.000000,\Ry:=0.000000),vel1,zoneval,Extruder\WObj:=Workobject_1;
MoveL RelTool (p1,38.000000,14.500000,18.230831,\Rx:=0.000000,\Ry:=0.000000),vel1,zoneval,Extruder\WObj:=Workobject_1;
MoveL RelTool (p1,38.500000,14.500000,18.279434,\Rx:=0.000000,\Ry:=0.000000),vel1,zoneval,Extruder\WObj:=Workobject_1;
MoveL RelTool (p1,39.000000,14.500000,18.328464,\Rx:=0.000000,\Ry:=0.000000),vel1,zoneval,Extruder\WObj:=Workobject_1;
MoveL RelTool (p1,39.500000,14.500000,18.372133,\Rx:=0.000000,\Ry:=0.000000),vel1,zoneval,Extruder\WObj:=Workobject_1;
MoveL RelTool (p1,40.000000,14.500000,18.401583,\Rx:=0.000000,\Ry:=0.000000),vel1,zoneval,Extruder\WObj:=Workobject_1;
MoveL RelTool (p1,40.500000,14.500000,18.431033,\Rx:=0.000000,\Ry:=0.000000),vel1,zoneval,Extruder\WObj:=Workobject_1;
MoveL RelTool (p1,41.000000,14.500000,18.458031,\Rx:=0.000000,\Ry:=0.000000),vel1,zoneval,Extruder\WObj:=Workobject_1;
MoveL RelTool (p1,41.500000,14.500000,18.472733,\Rx:=0.000000,\Ry:=0.000000),vel1,zoneval,Extruder\WObj:=Workobject_1;
MoveL RelTool (p1,42.000000,14.500000,18.483145,\Rx:=0.000000,\Ry:=0.000000),vel1,zoneval,Extruder\WObj:=Workobject_1;
MoveL RelTool (p1,42.500000,14.500000,18.493557,\Rx:=0.000000,\Ry:=0.000000),vel1,zoneval,Extruder\WObj:=Workobject_1;
MoveL RelTool (p1,43.000000,14.500000,18.497374,\Rx:=0.000000,\Ry:=0.000000),vel1,zoneval,Extruder\WObj:=Workobject_1;
MoveL RelTool (p1,43.500000,14.500000,18.488845,\Rx:=0.000000,\Ry:=0.000000),vel1,zoneval,Extruder\WObj:=Workobject_1;
MoveL RelTool (p1,44.000000,14.500000,18.480316,\Rx:=0.000000,\Ry:=0.000000),vel1,zoneval,Extruder\WObj:=Workobject_1;
MoveL RelTool (p1,44.500000,14.500000,18.470425,\Rx:=0.000000,\Ry:=0.000000),vel1,zoneval,Extruder\WObj:=Workobject_1;
MoveL RelTool (p1,45.000000,14.500000,18.448443,\Rx:=0.000000,\Ry:=0.000000),vel1,zoneval,Extruder\WObj:=Workobject_1;
MoveL RelTool (p1,45.500000,14.500000,18.420900,\Rx:=0.000000,\Ry:=0.000000),vel1,zoneval,Extruder\WObj:=Workobject_1;
MoveL RelTool (p1,46.000000,14.500000,18.393356,\Rx:=0.000000,\Ry:=0.000000),vel1,zoneval,Extruder\WObj:=Workobject_1;
MoveL RelTool (p1,46.500000,14.500000,18.360102,\Rx:=0.000000,\Ry:=0.000000),vel1,zoneval,Extruder\WObj:=Workobject_1;
MoveL RelTool (p1,47.000000,14.500000,18.313470,\Rx:=0.000000,\Ry:=0.000000),vel1,zoneval,Extruder\WObj:=Workobject_1;
MoveL RelTool (p1,47.500000,14.500000,18.266839,\Rx:=0.000000,\Ry:=0.000000),vel1,zoneval,Extruder\WObj:=Workobject_1;
MoveL RelTool (p1,48.000000,14.500000,18.219419,\Rx:=0.000000,\Ry:=0.000000),vel1,zoneval,Extruder\WObj:=Workobject_1;
MoveL RelTool (p1,48.500000,14.500000,18.160867,\Rx:=0.000000,\Ry:=0.000000),vel1,zoneval,Extruder\WObj:=Workobject_1;
MoveL RelTool (p1,49.000000,14.500000,18.094810,\Rx:=0.000000,\Ry:=0.000000),vel1,zoneval,Extruder\WObj:=Workobject_1;
MoveL RelTool (p1,49.500000,14.500000,18.028753,\Rx:=0.000000,\Ry:=0.000000),vel1,zoneval,Extruder\WObj:=Workobject_1;
MoveL RelTool (p1,50.000000,14.500000,17.952741,\Rx:=0.000000,\Ry:=0.000000),vel1,zoneval,Extruder\WObj:=Workobject_1;
MoveL RelTool (p1,50.500000,14.500000,17.866764,\Rx:=0.000000,\Ry:=0.000000),vel1,zoneval,Extruder\WObj:=Workobject_1;
MoveL RelTool (p1,51.000000,14.500000,17.780788,\Rx:=0.000000,\Ry:=0.000000),vel1,zoneval,Extruder\WObj:=Workobject_1;
MoveL RelTool (p1,51.500000,14.500000,17.695839,\Rx:=0.000000,\Ry:=0.000000),vel1,zoneval,Extruder\WObj:=Workobject_1;
MoveL RelTool (p1,52.000000,14.500000,17.590910,\Rx:=0.000000,\Ry:=0.000000),vel1,zoneval,Extruder\WObj:=Workobject_1;
MoveL RelTool (p1,52.500000,14.500000,17.484155,\Rx:=0.000000,\Ry:=0.000000),vel1,zoneval,Extruder\WObj:=Workobject_1;
MoveL RelTool (p1,53.000000,14.500000,17.375041,\Rx:=0.000000,\Ry:=0.000000),vel1,zoneval,Extruder\WObj:=Workobject_1;
MoveL RelTool (p1,53.500000,14.500000,17.246441,\Rx:=0.000000,\Ry:=0.000000),vel1,zoneval,Extruder\WObj:=Workobject_1;
MoveL RelTool (p1,54.000000,14.500000,17.117841,\Rx:=0.000000,\Ry:=0.000000),vel1,zoneval,Extruder\WObj:=Workobject_1;
MoveL RelTool (p1,54.500000,14.500000,16.992475,\Rx:=0.000000,\Ry:=0.000000),vel1,zoneval,Extruder\WObj:=Workobject_1;
MoveL RelTool (p1,55.000000,14.500000,16.847563,\Rx:=0.000000,\Ry:=0.000000),vel1,zoneval,Extruder\WObj:=Workobject_1;
MoveL RelTool (p1,55.500000,14.500000,16.695948,\Rx:=0.000000,\Ry:=0.000000),vel1,zoneval,Extruder\WObj:=Workobject_1;
MoveL RelTool (p1,56.000000,14.500000,16.542748,\Rx:=0.000000,\Ry:=0.000000),vel1,zoneval,Extruder\WObj:=Workobject_1;
MoveL RelTool (p1,56.500000,14.500000,16.372932,\Rx:=0.000000,\Ry:=0.000000),vel1,zoneval,Extruder\WObj:=Workobject_1;
MoveL RelTool (p1,57.000000,14.500000,16.197022,\Rx:=0.000000,\Ry:=0.000000),vel1,zoneval,Extruder\WObj:=Workobject_1;
MoveL RelTool (p1,57.500000,14.500000,16.018147,\Rx:=0.000000,\Ry:=0.000000),vel1,zoneval,Extruder\WObj:=Workobject_1;
MoveL RelTool (p1,58.000000,14.500000,15.816521,\Rx:=0.000000,\Ry:=0.000000),vel1,zoneval,Extruder\WObj:=Workobject_1;
MoveL RelTool (p1,58.500000,14.500000,15.614895,\Rx:=0.000000,\Ry:=0.000000),vel1,zoneval,Extruder\WObj:=Workobject_1;
MoveL RelTool (p1,59.000000,14.500000,15.404082,\Rx:=0.000000,\Ry:=0.000000),vel1,zoneval,Extruder\WObj:=Workobject_1;
MoveL RelTool (p1,59.500000,14.500000,15.174285,\Rx:=0.000000,\Ry:=0.000000),vel1,zoneval,Extruder\WObj:=Workobject_1;
MoveL RelTool (p1,60.000000,14.500000,14.939580,\Rx:=0.000000,\Ry:=0.000000),vel1,zoneval,Extruder\WObj:=Workobject_1;
MoveL RelTool (p1,60.500000,14.500000,14.678534,\Rx:=0.000000,\Ry:=0.000000),vel1,zoneval,Extruder\WObj:=Workobject_1;
MoveL RelTool (p1,61.000000,14.500000,14.418869,\Rx:=0.000000,\Ry:=0.000000),vel1,zoneval,Extruder\WObj:=Workobject_1;
MoveL RelTool (p1,61.500000,14.500000,14.134258,\Rx:=0.000000,\Ry:=0.000000),vel1,zoneval,Extruder\WObj:=Workobject_1;
MoveL RelTool (p1,62.000000,14.500000,13.838283,\Rx:=0.000000,\Ry:=0.000000),vel1,zoneval,Extruder\WObj:=Workobject_1;
MoveL RelTool (p1,62.500000,14.500000,13.514668,\Rx:=0.000000,\Ry:=0.000000),vel1,zoneval,Extruder\WObj:=Workobject_1;
MoveL RelTool (p1,63.000000,14.500000,13.179296,\Rx:=0.000000,\Ry:=0.000000),vel1,zoneval,Extruder\WObj:=Workobject_1;
MoveL RelTool (p1,63.500000,14.500000,12.806154,\Rx:=0.000000,\Ry:=0.000000),vel1,zoneval,Extruder\WObj:=Workobject_1;
MoveL RelTool (p1,64.000000,14.500000,12.421949,\Rx:=0.000000,\Ry:=0.000000),vel1,zoneval,Extruder\WObj:=Workobject_1;
MoveL RelTool (p1,64.500000,14.500000,11.989135,\Rx:=0.000000,\Ry:=0.000000),vel1,zoneval,Extruder\WObj:=Workobject_1;
MoveL RelTool (p1,65.000000,14.500000,11.515128,\Rx:=0.000000,\Ry:=0.000000),vel1,zoneval,Extruder\WObj:=Workobject_1;
MoveL RelTool (p1,65.500000,14.500000,11.006720,\Rx:=0.000000,\Ry:=0.000000),vel1,zoneval,Extruder\WObj:=Workobject_1;
MoveL RelTool (p1,66.000000,14.500000,10.426294,\Rx:=0.000000,\Ry:=0.000000),vel1,zoneval,Extruder\WObj:=Workobject_1;
MoveL RelTool (p1,66.500000,14.500000,9.763981,\Rx:=0.000000,\Ry:=0.000000),vel1,zoneval,Extruder\WObj:=Workobject_1;
MoveL RelTool (p1,67.000000,14.500000,9.225973,\Rx:=0.000000,\Ry:=0.000000),vel1,zoneval,Extruder\WObj:=Workobject_1;
MoveL RelTool (p1,67.500000,14.500000,8.874086,\Rx:=0.000000,\Ry:=0.000000),vel1,zoneval,Extruder\WObj:=Workobject_1;
MoveL RelTool (p1,68.000000,14.500000,8.652682,\Rx:=0.000000,\Ry:=0.000000),vel1,zoneval,Extruder\WObj:=Workobject_1;
MoveL RelTool (p1,68.500000,14.500000,8.535785,\Rx:=0.000000,\Ry:=0.000000),vel1,zoneval,Extruder\WObj:=Workobject_1;
MoveL RelTool (p1,69.000000,14.500000,8.500000,\Rx:=0.000000,\Ry:=0.000000),vel1,zoneval,Extruder\WObj:=Workobject_1;
MoveL RelTool (p1,69.500000,14.500000,8.500000,\Rx:=0.000000,\Ry:=0.000000),vel1,zoneval,Extruder\WObj:=Workobject_1;
MoveL RelTool (p1,70.000000,14.500000,8.500000,\Rx:=0.000000,\Ry:=0.000000),vel1,zoneval,Extruder\WObj:=Workobject_1;
MoveL RelTool (p1,70.500000,14.500000,8.500000,\Rx:=0.000000,\Ry:=0.000000),vel1,zoneval,Extruder\WObj:=Workobject_1;
MoveL RelTool (p1,71.000000,14.500000,8.500000,\Rx:=0.000000,\Ry:=0.000000),vel1,zoneval,Extruder\WObj:=Workobject_1;
MoveL RelTool (p1,71.500000,14.500000,8.500000,\Rx:=0.000000,\Ry:=0.000000),vel1,zoneval,Extruder\WObj:=Workobject_1;
MoveL RelTool (p1,72.000000,14.500000,8.500000,\Rx:=0.000000,\Ry:=0.000000),vel1,zoneval,Extruder\WObj:=Workobject_1;
MoveL RelTool (p1,72.500000,14.500000,8.500000,\Rx:=0.000000,\Ry:=0.000000),vel1,zoneval,Extruder\WObj:=Workobject_1;
MoveL RelTool (p1,73.000000,14.500000,8.500000,\Rx:=0.000000,\Ry:=0.000000),vel1,zoneval,Extruder\WObj:=Workobject_1;
MoveL RelTool (p1,73.500000,14.500000,8.500000,\Rx:=0.000000,\Ry:=0.000000),vel1,zoneval,Extruder\WObj:=Workobject_1;
MoveL RelTool (p1,74.000000,14.500000,8.500000,\Rx:=0.000000,\Ry:=0.000000),vel1,zoneval,Extruder\WObj:=Workobject_1;
MoveL RelTool (p1,74.500000,14.500000,8.500000,\Rx:=0.000000,\Ry:=0.000000),vel1,zoneval,Extruder\WObj:=Workobject_1;
MoveL RelTool (p1,75.000000,14.500000,8.500000,\Rx:=0.000000,\Ry:=0.000000),vel1,zoneval,Extruder\WObj:=Workobject_1;
MoveL RelTool (p1,75.500000,14.500000,8.500000,\Rx:=0.000000,\Ry:=0.000000),vel1,zoneval,Extruder\WObj:=Workobject_1;
MoveL RelTool (p1,76.000000,14.500000,8.500000,\Rx:=0.000000,\Ry:=0.000000),vel1,zoneval,Extruder\WObj:=Workobject_1;
MoveL RelTool (p1,76.500000,14.500000,8.500000,\Rx:=0.000000,\Ry:=0.000000),vel1,zoneval,Extruder\WObj:=Workobject_1;
MoveL RelTool (p1,77.000000,14.500000,8.500000,\Rx:=0.000000,\Ry:=0.000000),vel1,zoneval,Extruder\WObj:=Workobject_1;
MoveL RelTool (p1,77.500000,14.500000,8.500000,\Rx:=0.000000,\Ry:=0.000000),vel1,zoneval,Extruder\WObj:=Workobject_1;
MoveL RelTool (p1,78.000000,14.500000,8.500000,\Rx:=0.000000,\Ry:=0.000000),vel1,zoneval,Extruder\WObj:=Workobject_1;
MoveL RelTool (p1,78.500000,14.500000,8.500000,\Rx:=0.000000,\Ry:=0.000000),vel1,zoneval,Extruder\WObj:=Workobject_1;
MoveL RelTool (p1,79.000000,14.500000,8.500000,\Rx:=0.000000,\Ry:=0.000000),vel1,zoneval,Extruder\WObj:=Workobject_1;
MoveL RelTool (p1,79.500000,14.500000,8.500000,\Rx:=0.000000,\Ry:=0.000000),vel1,zoneval,Extruder\WObj:=Workobject_1;
MoveL RelTool (p1,80.000000,14.500000,8.500000,\Rx:=0.000000,\Ry:=0.000000),vel1,zoneval,Extruder\WObj:=Workobject_1;
MoveL RelTool (p1,80.500000,14.500000,8.500000,\Rx:=0.000000,\Ry:=0.000000),vel1,zoneval,Extruder\WObj:=Workobject_1;
MoveL RelTool (p1,81.000000,14.500000,8.500000,\Rx:=0.000000,\Ry:=0.000000),vel1,zoneval,Extruder\WObj:=Workobject_1;
MoveL RelTool (p1,81.500000,14.500000,8.500000,\Rx:=0.000000,\Ry:=0.000000),vel1,zoneval,Extruder\WObj:=Workobject_1;
MoveL RelTool (p1,82.000000,14.500000,8.500000,\Rx:=0.000000,\Ry:=0.000000),vel1,zoneval,Extruder\WObj:=Workobject_1;
MoveL RelTool (p1,82.000000,15.000000,8.500000,\Rx:=0.000000,\Ry:=0.000000),vel1,zoneval,Extruder\WObj:=Workobject_1;
MoveL RelTool (p1,81.500000,15.000000,8.500000,\Rx:=0.000000,\Ry:=0.000000),vel1,zoneval,Extruder\WObj:=Workobject_1;
MoveL RelTool (p1,81.000000,15.000000,8.500000,\Rx:=0.000000,\Ry:=0.000000),vel1,zoneval,Extruder\WObj:=Workobject_1;
MoveL RelTool (p1,80.500000,15.000000,8.500000,\Rx:=0.000000,\Ry:=0.000000),vel1,zoneval,Extruder\WObj:=Workobject_1;
MoveL RelTool (p1,80.000000,15.000000,8.500000,\Rx:=0.000000,\Ry:=0.000000),vel1,zoneval,Extruder\WObj:=Workobject_1;
MoveL RelTool (p1,79.500000,15.000000,8.500000,\Rx:=0.000000,\Ry:=0.000000),vel1,zoneval,Extruder\WObj:=Workobject_1;
MoveL RelTool (p1,79.000000,15.000000,8.500000,\Rx:=0.000000,\Ry:=0.000000),vel1,zoneval,Extruder\WObj:=Workobject_1;
MoveL RelTool (p1,78.500000,15.000000,8.500000,\Rx:=0.000000,\Ry:=0.000000),vel1,zoneval,Extruder\WObj:=Workobject_1;
MoveL RelTool (p1,78.000000,15.000000,8.500000,\Rx:=0.000000,\Ry:=0.000000),vel1,zoneval,Extruder\WObj:=Workobject_1;
MoveL RelTool (p1,77.500000,15.000000,8.500000,\Rx:=0.000000,\Ry:=0.000000),vel1,zoneval,Extruder\WObj:=Workobject_1;
MoveL RelTool (p1,77.000000,15.000000,8.500000,\Rx:=0.000000,\Ry:=0.000000),vel1,zoneval,Extruder\WObj:=Workobject_1;
MoveL RelTool (p1,76.500000,15.000000,8.500000,\Rx:=0.000000,\Ry:=0.000000),vel1,zoneval,Extruder\WObj:=Workobject_1;
MoveL RelTool (p1,76.000000,15.000000,8.500000,\Rx:=0.000000,\Ry:=0.000000),vel1,zoneval,Extruder\WObj:=Workobject_1;
MoveL RelTool (p1,75.500000,15.000000,8.500000,\Rx:=0.000000,\Ry:=0.000000),vel1,zoneval,Extruder\WObj:=Workobject_1;
MoveL RelTool (p1,75.000000,15.000000,8.500000,\Rx:=0.000000,\Ry:=0.000000),vel1,zoneval,Extruder\WObj:=Workobject_1;
MoveL RelTool (p1,74.500000,15.000000,8.500000,\Rx:=0.000000,\Ry:=0.000000),vel1,zoneval,Extruder\WObj:=Workobject_1;
MoveL RelTool (p1,74.000000,15.000000,8.500000,\Rx:=0.000000,\Ry:=0.000000),vel1,zoneval,Extruder\WObj:=Workobject_1;
MoveL RelTool (p1,73.500000,15.000000,8.500000,\Rx:=0.000000,\Ry:=0.000000),vel1,zoneval,Extruder\WObj:=Workobject_1;
MoveL RelTool (p1,73.000000,15.000000,8.500000,\Rx:=0.000000,\Ry:=0.000000),vel1,zoneval,Extruder\WObj:=Workobject_1;
MoveL RelTool (p1,72.500000,15.000000,8.500000,\Rx:=0.000000,\Ry:=0.000000),vel1,zoneval,Extruder\WObj:=Workobject_1;
MoveL RelTool (p1,72.000000,15.000000,8.500000,\Rx:=0.000000,\Ry:=0.000000),vel1,zoneval,Extruder\WObj:=Workobject_1;
MoveL RelTool (p1,71.500000,15.000000,8.500000,\Rx:=0.000000,\Ry:=0.000000),vel1,zoneval,Extruder\WObj:=Workobject_1;
MoveL RelTool (p1,71.000000,15.000000,8.500000,\Rx:=0.000000,\Ry:=0.000000),vel1,zoneval,Extruder\WObj:=Workobject_1;
MoveL RelTool (p1,70.500000,15.000000,8.500000,\Rx:=0.000000,\Ry:=0.000000),vel1,zoneval,Extruder\WObj:=Workobject_1;
MoveL RelTool (p1,70.000000,15.000000,8.500000,\Rx:=0.000000,\Ry:=0.000000),vel1,zoneval,Extruder\WObj:=Workobject_1;
MoveL RelTool (p1,69.500000,15.000000,8.500000,\Rx:=0.000000,\Ry:=0.000000),vel1,zoneval,Extruder\WObj:=Workobject_1;
MoveL RelTool (p1,69.000000,15.000000,8.500000,\Rx:=0.000000,\Ry:=0.000000),vel1,zoneval,Extruder\WObj:=Workobject_1;
MoveL RelTool (p1,68.500000,15.000000,8.535785,\Rx:=0.000000,\Ry:=0.000000),vel1,zoneval,Extruder\WObj:=Workobject_1;
MoveL RelTool (p1,68.000000,15.000000,8.652682,\Rx:=0.000000,\Ry:=0.000000),vel1,zoneval,Extruder\WObj:=Workobject_1;
MoveL RelTool (p1,67.500000,15.000000,8.874086,\Rx:=0.000000,\Ry:=0.000000),vel1,zoneval,Extruder\WObj:=Workobject_1;
MoveL RelTool (p1,67.000000,15.000000,9.225973,\Rx:=0.000000,\Ry:=0.000000),vel1,zoneval,Extruder\WObj:=Workobject_1;
MoveL RelTool (p1,66.500000,15.000000,9.763981,\Rx:=0.000000,\Ry:=0.000000),vel1,zoneval,Extruder\WObj:=Workobject_1;
MoveL RelTool (p1,66.000000,15.000000,10.427806,\Rx:=0.000000,\Ry:=0.000000),vel1,zoneval,Extruder\WObj:=Workobject_1;
MoveL RelTool (p1,65.500000,15.000000,11.006360,\Rx:=0.000000,\Ry:=0.000000),vel1,zoneval,Extruder\WObj:=Workobject_1;
MoveL RelTool (p1,65.000000,15.000000,11.516294,\Rx:=0.000000,\Ry:=0.000000),vel1,zoneval,Extruder\WObj:=Workobject_1;
MoveL RelTool (p1,64.500000,15.000000,11.988727,\Rx:=0.000000,\Ry:=0.000000),vel1,zoneval,Extruder\WObj:=Workobject_1;
MoveL RelTool (p1,64.000000,15.000000,12.421541,\Rx:=0.000000,\Ry:=0.000000),vel1,zoneval,Extruder\WObj:=Workobject_1;
MoveL RelTool (p1,63.500000,15.000000,12.806452,\Rx:=0.000000,\Ry:=0.000000),vel1,zoneval,Extruder\WObj:=Workobject_1;
MoveL RelTool (p1,63.000000,15.000000,13.179092,\Rx:=0.000000,\Ry:=0.000000),vel1,zoneval,Extruder\WObj:=Workobject_1;
MoveL RelTool (p1,62.500000,15.000000,13.514464,\Rx:=0.000000,\Ry:=0.000000),vel1,zoneval,Extruder\WObj:=Workobject_1;
MoveL RelTool (p1,62.000000,15.000000,13.838119,\Rx:=0.000000,\Ry:=0.000000),vel1,zoneval,Extruder\WObj:=Workobject_1;
MoveL RelTool (p1,61.500000,15.000000,14.134095,\Rx:=0.000000,\Ry:=0.000000),vel1,zoneval,Extruder\WObj:=Workobject_1;
MoveL RelTool (p1,61.000000,15.000000,14.419171,\Rx:=0.000000,\Ry:=0.000000),vel1,zoneval,Extruder\WObj:=Workobject_1;
MoveL RelTool (p1,60.500000,15.000000,14.679885,\Rx:=0.000000,\Ry:=0.000000),vel1,zoneval,Extruder\WObj:=Workobject_1;
MoveL RelTool (p1,60.000000,15.000000,14.940931,\Rx:=0.000000,\Ry:=0.000000),vel1,zoneval,Extruder\WObj:=Workobject_1;
MoveL RelTool (p1,59.500000,15.000000,15.173961,\Rx:=0.000000,\Ry:=0.000000),vel1,zoneval,Extruder\WObj:=Workobject_1;
MoveL RelTool (p1,59.000000,15.000000,15.403758,\Rx:=0.000000,\Ry:=0.000000),vel1,zoneval,Extruder\WObj:=Workobject_1;
MoveL RelTool (p1,58.500000,15.000000,15.615386,\Rx:=0.000000,\Ry:=0.000000),vel1,zoneval,Extruder\WObj:=Workobject_1;
MoveL RelTool (p1,58.000000,15.000000,15.817012,\Rx:=0.000000,\Ry:=0.000000),vel1,zoneval,Extruder\WObj:=Workobject_1;
MoveL RelTool (p1,57.500000,15.000000,16.018639,\Rx:=0.000000,\Ry:=0.000000),vel1,zoneval,Extruder\WObj:=Workobject_1;
MoveL RelTool (p1,57.000000,15.000000,16.196753,\Rx:=0.000000,\Ry:=0.000000),vel1,zoneval,Extruder\WObj:=Workobject_1;
MoveL RelTool (p1,56.500000,15.000000,16.372663,\Rx:=0.000000,\Ry:=0.000000),vel1,zoneval,Extruder\WObj:=Workobject_1;
MoveL RelTool (p1,56.000000,15.000000,16.543721,\Rx:=0.000000,\Ry:=0.000000),vel1,zoneval,Extruder\WObj:=Workobject_1;
MoveL RelTool (p1,55.500000,15.000000,16.695963,\Rx:=0.000000,\Ry:=0.000000),vel1,zoneval,Extruder\WObj:=Workobject_1;
MoveL RelTool (p1,55.000000,15.000000,16.847578,\Rx:=0.000000,\Ry:=0.000000),vel1,zoneval,Extruder\WObj:=Workobject_1;
MoveL RelTool (p1,54.500000,15.000000,16.992526,\Rx:=0.000000,\Ry:=0.000000),vel1,zoneval,Extruder\WObj:=Workobject_1;
MoveL RelTool (p1,54.000000,15.000000,17.119535,\Rx:=0.000000,\Ry:=0.000000),vel1,zoneval,Extruder\WObj:=Workobject_1;
MoveL RelTool (p1,53.500000,15.000000,17.248135,\Rx:=0.000000,\Ry:=0.000000),vel1,zoneval,Extruder\WObj:=Workobject_1;
MoveL RelTool (p1,53.000000,15.000000,17.376735,\Rx:=0.000000,\Ry:=0.000000),vel1,zoneval,Extruder\WObj:=Workobject_1;
MoveL RelTool (p1,52.500000,15.000000,17.483908,\Rx:=0.000000,\Ry:=0.000000),vel1,zoneval,Extruder\WObj:=Workobject_1;
MoveL RelTool (p1,52.000000,15.000000,17.590663,\Rx:=0.000000,\Ry:=0.000000),vel1,zoneval,Extruder\WObj:=Workobject_1;
MoveL RelTool (p1,51.500000,15.000000,17.696345,\Rx:=0.000000,\Ry:=0.000000),vel1,zoneval,Extruder\WObj:=Workobject_1;
MoveL RelTool (p1,51.000000,15.000000,17.781625,\Rx:=0.000000,\Ry:=0.000000),vel1,zoneval,Extruder\WObj:=Workobject_1;
MoveL RelTool (p1,50.500000,15.000000,17.867602,\Rx:=0.000000,\Ry:=0.000000),vel1,zoneval,Extruder\WObj:=Workobject_1;
MoveL RelTool (p1,50.000000,15.000000,17.953578,\Rx:=0.000000,\Ry:=0.000000),vel1,zoneval,Extruder\WObj:=Workobject_1;
MoveL RelTool (p1,49.500000,15.000000,18.028437,\Rx:=0.000000,\Ry:=0.000000),vel1,zoneval,Extruder\WObj:=Workobject_1;
MoveL RelTool (p1,49.000000,15.000000,18.094494,\Rx:=0.000000,\Ry:=0.000000),vel1,zoneval,Extruder\WObj:=Workobject_1;
MoveL RelTool (p1,48.500000,15.000000,18.160551,\Rx:=0.000000,\Ry:=0.000000),vel1,zoneval,Extruder\WObj:=Workobject_1;
MoveL RelTool (p1,48.000000,15.000000,18.220248,\Rx:=0.000000,\Ry:=0.000000),vel1,zoneval,Extruder\WObj:=Workobject_1;
MoveL RelTool (p1,47.500000,15.000000,18.267072,\Rx:=0.000000,\Ry:=0.000000),vel1,zoneval,Extruder\WObj:=Workobject_1;
MoveL RelTool (p1,47.000000,15.000000,18.313704,\Rx:=0.000000,\Ry:=0.000000),vel1,zoneval,Extruder\WObj:=Workobject_1;
MoveL RelTool (p1,46.500000,15.000000,18.360335,\Rx:=0.000000,\Ry:=0.000000),vel1,zoneval,Extruder\WObj:=Workobject_1;
MoveL RelTool (p1,46.000000,15.000000,18.393186,\Rx:=0.000000,\Ry:=0.000000),vel1,zoneval,Extruder\WObj:=Workobject_1;
MoveL RelTool (p1,45.500000,15.000000,18.420730,\Rx:=0.000000,\Ry:=0.000000),vel1,zoneval,Extruder\WObj:=Workobject_1;
MoveL RelTool (p1,45.000000,15.000000,18.448274,\Rx:=0.000000,\Ry:=0.000000),vel1,zoneval,Extruder\WObj:=Workobject_1;
MoveL RelTool (p1,44.500000,15.000000,18.471400,\Rx:=0.000000,\Ry:=0.000000),vel1,zoneval,Extruder\WObj:=Workobject_1;
MoveL RelTool (p1,44.000000,15.000000,18.480187,\Rx:=0.000000,\Ry:=0.000000),vel1,zoneval,Extruder\WObj:=Workobject_1;
MoveL RelTool (p1,43.500000,15.000000,18.488716,\Rx:=0.000000,\Ry:=0.000000),vel1,zoneval,Extruder\WObj:=Workobject_1;
MoveL RelTool (p1,43.000000,15.000000,18.497245,\Rx:=0.000000,\Ry:=0.000000),vel1,zoneval,Extruder\WObj:=Workobject_1;
MoveL RelTool (p1,42.500000,15.000000,18.493401,\Rx:=0.000000,\Ry:=0.000000),vel1,zoneval,Extruder\WObj:=Workobject_1;
MoveL RelTool (p1,42.000000,15.000000,18.482989,\Rx:=0.000000,\Ry:=0.000000),vel1,zoneval,Extruder\WObj:=Workobject_1;
MoveL RelTool (p1,41.500000,15.000000,18.472577,\Rx:=0.000000,\Ry:=0.000000),vel1,zoneval,Extruder\WObj:=Workobject_1;
MoveL RelTool (p1,41.000000,15.000000,18.459000,\Rx:=0.000000,\Ry:=0.000000),vel1,zoneval,Extruder\WObj:=Workobject_1;
MoveL RelTool (p1,40.500000,15.000000,18.430881,\Rx:=0.000000,\Ry:=0.000000),vel1,zoneval,Extruder\WObj:=Workobject_1;
MoveL RelTool (p1,40.000000,15.000000,18.401431,\Rx:=0.000000,\Ry:=0.000000),vel1,zoneval,Extruder\WObj:=Workobject_1;
MoveL RelTool (p1,39.500000,15.000000,18.371981,\Rx:=0.000000,\Ry:=0.000000),vel1,zoneval,Extruder\WObj:=Workobject_1;
MoveL RelTool (p1,39.000000,15.000000,18.329277,\Rx:=0.000000,\Ry:=0.000000),vel1,zoneval,Extruder\WObj:=Workobject_1;
MoveL RelTool (p1,38.500000,15.000000,18.280674,\Rx:=0.000000,\Ry:=0.000000),vel1,zoneval,Extruder\WObj:=Workobject_1;
MoveL RelTool (p1,38.000000,15.000000,18.232071,\Rx:=0.000000,\Ry:=0.000000),vel1,zoneval,Extruder\WObj:=Workobject_1;
MoveL RelTool (p1,37.500000,15.000000,18.183468,\Rx:=0.000000,\Ry:=0.000000),vel1,zoneval,Extruder\WObj:=Workobject_1;
MoveL RelTool (p1,37.000000,15.000000,18.117521,\Rx:=0.000000,\Ry:=0.000000),vel1,zoneval,Extruder\WObj:=Workobject_1;
MoveL RelTool (p1,36.500000,15.000000,18.049256,\Rx:=0.000000,\Ry:=0.000000),vel1,zoneval,Extruder\WObj:=Workobject_1;
MoveL RelTool (p1,36.000000,15.000000,17.980992,\Rx:=0.000000,\Ry:=0.000000),vel1,zoneval,Extruder\WObj:=Workobject_1;
MoveL RelTool (p1,35.500000,15.000000,17.898537,\Rx:=0.000000,\Ry:=0.000000),vel1,zoneval,Extruder\WObj:=Workobject_1;
MoveL RelTool (p1,35.000000,15.000000,17.809963,\Rx:=0.000000,\Ry:=0.000000),vel1,zoneval,Extruder\WObj:=Workobject_1;
MoveL RelTool (p1,34.500000,15.000000,17.721390,\Rx:=0.000000,\Ry:=0.000000),vel1,zoneval,Extruder\WObj:=Workobject_1;
MoveL RelTool (p1,34.000000,15.000000,17.629837,\Rx:=0.000000,\Ry:=0.000000),vel1,zoneval,Extruder\WObj:=Workobject_1;
MoveL RelTool (p1,33.500000,15.000000,17.519910,\Rx:=0.000000,\Ry:=0.000000),vel1,zoneval,Extruder\WObj:=Workobject_1;
MoveL RelTool (p1,33.000000,15.000000,17.409983,\Rx:=0.000000,\Ry:=0.000000),vel1,zoneval,Extruder\WObj:=Workobject_1;
MoveL RelTool (p1,32.500000,15.000000,17.297270,\Rx:=0.000000,\Ry:=0.000000),vel1,zoneval,Extruder\WObj:=Workobject_1;
MoveL RelTool (p1,32.000000,15.000000,17.166480,\Rx:=0.000000,\Ry:=0.000000),vel1,zoneval,Extruder\WObj:=Workobject_1;
MoveL RelTool (p1,31.500000,15.000000,17.034076,\Rx:=0.000000,\Ry:=0.000000),vel1,zoneval,Extruder\WObj:=Workobject_1;
MoveL RelTool (p1,31.000000,15.000000,16.901672,\Rx:=0.000000,\Ry:=0.000000),vel1,zoneval,Extruder\WObj:=Workobject_1;
MoveL RelTool (p1,30.500000,15.000000,16.747980,\Rx:=0.000000,\Ry:=0.000000),vel1,zoneval,Extruder\WObj:=Workobject_1;
MoveL RelTool (p1,30.000000,15.000000,16.591911,\Rx:=0.000000,\Ry:=0.000000),vel1,zoneval,Extruder\WObj:=Workobject_1;
MoveL RelTool (p1,29.500000,15.000000,16.434130,\Rx:=0.000000,\Ry:=0.000000),vel1,zoneval,Extruder\WObj:=Workobject_1;
MoveL RelTool (p1,29.000000,15.000000,16.256339,\Rx:=0.000000,\Ry:=0.000000),vel1,zoneval,Extruder\WObj:=Workobject_1;
MoveL RelTool (p1,28.500000,15.000000,16.075339,\Rx:=0.000000,\Ry:=0.000000),vel1,zoneval,Extruder\WObj:=Workobject_1;
MoveL RelTool (p1,28.000000,15.000000,15.890122,\Rx:=0.000000,\Ry:=0.000000),vel1,zoneval,Extruder\WObj:=Workobject_1;
MoveL RelTool (p1,27.500000,15.000000,15.682286,\Rx:=0.000000,\Ry:=0.000000),vel1,zoneval,Extruder\WObj:=Workobject_1;
MoveL RelTool (p1,27.000000,15.000000,15.474450,\Rx:=0.000000,\Ry:=0.000000),vel1,zoneval,Extruder\WObj:=Workobject_1;
MoveL RelTool (p1,26.500000,15.000000,15.254025,\Rx:=0.000000,\Ry:=0.000000),vel1,zoneval,Extruder\WObj:=Workobject_1;
MoveL RelTool (p1,26.000000,15.000000,15.016273,\Rx:=0.000000,\Ry:=0.000000),vel1,zoneval,Extruder\WObj:=Workobject_1;
MoveL RelTool (p1,25.500000,15.000000,14.775697,\Rx:=0.000000,\Ry:=0.000000),vel1,zoneval,Extruder\WObj:=Workobject_1;
MoveL RelTool (p1,25.000000,15.000000,14.505025,\Rx:=0.000000,\Ry:=0.000000),vel1,zoneval,Extruder\WObj:=Workobject_1;
MoveL RelTool (p1,24.500000,15.000000,14.233824,\Rx:=0.000000,\Ry:=0.000000),vel1,zoneval,Extruder\WObj:=Workobject_1;
MoveL RelTool (p1,24.000000,15.000000,13.936452,\Rx:=0.000000,\Ry:=0.000000),vel1,zoneval,Extruder\WObj:=Workobject_1;
MoveL RelTool (p1,23.500000,15.000000,13.627755,\Rx:=0.000000,\Ry:=0.000000),vel1,zoneval,Extruder\WObj:=Workobject_1;
MoveL RelTool (p1,23.000000,15.000000,13.289350,\Rx:=0.000000,\Ry:=0.000000),vel1,zoneval,Extruder\WObj:=Workobject_1;
MoveL RelTool (p1,22.500000,15.000000,12.938419,\Rx:=0.000000,\Ry:=0.000000),vel1,zoneval,Extruder\WObj:=Workobject_1;
MoveL RelTool (p1,22.000000,15.000000,12.548116,\Rx:=0.000000,\Ry:=0.000000),vel1,zoneval,Extruder\WObj:=Workobject_1;
MoveL RelTool (p1,21.500000,15.000000,12.140834,\Rx:=0.000000,\Ry:=0.000000),vel1,zoneval,Extruder\WObj:=Workobject_1;
MoveL RelTool (p1,21.000000,15.000000,11.682869,\Rx:=0.000000,\Ry:=0.000000),vel1,zoneval,Extruder\WObj:=Workobject_1;
MoveL RelTool (p1,20.500000,15.000000,11.179474,\Rx:=0.000000,\Ry:=0.000000),vel1,zoneval,Extruder\WObj:=Workobject_1;
MoveL RelTool (p1,20.000000,15.000000,10.624916,\Rx:=0.000000,\Ry:=0.000000),vel1,zoneval,Extruder\WObj:=Workobject_1;
MoveL RelTool (p1,19.500000,15.000000,9.992651,\Rx:=0.000000,\Ry:=0.000000),vel1,zoneval,Extruder\WObj:=Workobject_1;
MoveL RelTool (p1,19.000000,15.000000,9.374813,\Rx:=0.000000,\Ry:=0.000000),vel1,zoneval,Extruder\WObj:=Workobject_1;
MoveL RelTool (p1,18.500000,15.000000,8.980296,\Rx:=0.000000,\Ry:=0.000000),vel1,zoneval,Extruder\WObj:=Workobject_1;
MoveL RelTool (p1,18.000000,15.000000,8.722633,\Rx:=0.000000,\Ry:=0.000000),vel1,zoneval,Extruder\WObj:=Workobject_1;
MoveL RelTool (p1,17.500000,15.000000,8.570628,\Rx:=0.000000,\Ry:=0.000000),vel1,zoneval,Extruder\WObj:=Workobject_1;
MoveL RelTool (p1,17.000000,15.000000,8.508911,\Rx:=0.000000,\Ry:=0.000000),vel1,zoneval,Extruder\WObj:=Workobject_1;
MoveL RelTool (p1,16.500000,15.000000,8.500000,\Rx:=0.000000,\Ry:=0.000000),vel1,zoneval,Extruder\WObj:=Workobject_1;
MoveL RelTool (p1,16.000000,15.000000,8.500000,\Rx:=0.000000,\Ry:=0.000000),vel1,zoneval,Extruder\WObj:=Workobject_1;
MoveL RelTool (p1,15.500000,15.000000,8.500000,\Rx:=0.000000,\Ry:=0.000000),vel1,zoneval,Extruder\WObj:=Workobject_1;
MoveL RelTool (p1,15.000000,15.000000,8.500000,\Rx:=0.000000,\Ry:=0.000000),vel1,zoneval,Extruder\WObj:=Workobject_1;
MoveL RelTool (p1,14.500000,15.000000,8.500000,\Rx:=0.000000,\Ry:=0.000000),vel1,zoneval,Extruder\WObj:=Workobject_1;
MoveL RelTool (p1,14.000000,15.000000,8.500000,\Rx:=0.000000,\Ry:=0.000000),vel1,zoneval,Extruder\WObj:=Workobject_1;
MoveL RelTool (p1,13.500000,15.000000,8.500000,\Rx:=0.000000,\Ry:=0.000000),vel1,zoneval,Extruder\WObj:=Workobject_1;
MoveL RelTool (p1,13.000000,15.000000,8.500000,\Rx:=0.000000,\Ry:=0.000000),vel1,zoneval,Extruder\WObj:=Workobject_1;
MoveL RelTool (p1,12.500000,15.000000,8.500000,\Rx:=0.000000,\Ry:=0.000000),vel1,zoneval,Extruder\WObj:=Workobject_1;
MoveL RelTool (p1,12.000000,15.000000,8.500000,\Rx:=0.000000,\Ry:=0.000000),vel1,zoneval,Extruder\WObj:=Workobject_1;
MoveL RelTool (p1,11.500000,15.000000,8.500000,\Rx:=0.000000,\Ry:=0.000000),vel1,zoneval,Extruder\WObj:=Workobject_1;
MoveL RelTool (p1,11.000000,15.000000,8.500000,\Rx:=0.000000,\Ry:=0.000000),vel1,zoneval,Extruder\WObj:=Workobject_1;
MoveL RelTool (p1,10.500000,15.000000,8.500000,\Rx:=0.000000,\Ry:=0.000000),vel1,zoneval,Extruder\WObj:=Workobject_1;
MoveL RelTool (p1,10.000000,15.000000,8.500000,\Rx:=0.000000,\Ry:=0.000000),vel1,zoneval,Extruder\WObj:=Workobject_1;
MoveL RelTool (p1,9.500000,15.000000,8.500000,\Rx:=0.000000,\Ry:=0.000000),vel1,zoneval,Extruder\WObj:=Workobject_1;
MoveL RelTool (p1,9.000000,15.000000,8.500000,\Rx:=0.000000,\Ry:=0.000000),vel1,zoneval,Extruder\WObj:=Workobject_1;
MoveL RelTool (p1,8.500000,15.000000,8.500000,\Rx:=0.000000,\Ry:=0.000000),vel1,zoneval,Extruder\WObj:=Workobject_1;
MoveL RelTool (p1,8.000000,15.000000,8.500000,\Rx:=0.000000,\Ry:=0.000000),vel1,zoneval,Extruder\WObj:=Workobject_1;
MoveL RelTool (p1,7.500000,15.000000,8.500000,\Rx:=0.000000,\Ry:=0.000000),vel1,zoneval,Extruder\WObj:=Workobject_1;
MoveL RelTool (p1,7.000000,15.000000,8.500000,\Rx:=0.000000,\Ry:=0.000000),vel1,zoneval,Extruder\WObj:=Workobject_1;
MoveL RelTool (p1,6.500000,15.000000,8.500000,\Rx:=0.000000,\Ry:=0.000000),vel1,zoneval,Extruder\WObj:=Workobject_1;
MoveL RelTool (p1,6.000000,15.000000,8.500000,\Rx:=0.000000,\Ry:=0.000000),vel1,zoneval,Extruder\WObj:=Workobject_1;
MoveL RelTool (p1,5.500000,15.000000,8.500000,\Rx:=0.000000,\Ry:=0.000000),vel1,zoneval,Extruder\WObj:=Workobject_1;
MoveL RelTool (p1,5.000000,15.000000,8.500000,\Rx:=0.000000,\Ry:=0.000000),vel1,zoneval,Extruder\WObj:=Workobject_1;
MoveL RelTool (p1,4.500000,15.000000,8.500000,\Rx:=0.000000,\Ry:=0.000000),vel1,zoneval,Extruder\WObj:=Workobject_1;
MoveL RelTool (p1,4.000000,15.000000,8.500000,\Rx:=0.000000,\Ry:=0.000000),vel1,zoneval,Extruder\WObj:=Workobject_1;
MoveL RelTool (p1,3.500000,15.000000,8.500000,\Rx:=0.000000,\Ry:=0.000000),vel1,zoneval,Extruder\WObj:=Workobject_1;
MoveL RelTool (p1,3.500000,15.500000,8.500000,\Rx:=0.000000,\Ry:=0.000000),vel1,zoneval,Extruder\WObj:=Workobject_1;
MoveL RelTool (p1,4.000000,15.500000,8.500000,\Rx:=0.000000,\Ry:=0.000000),vel1,zoneval,Extruder\WObj:=Workobject_1;
MoveL RelTool (p1,4.500000,15.500000,8.500000,\Rx:=0.000000,\Ry:=0.000000),vel1,zoneval,Extruder\WObj:=Workobject_1;
MoveL RelTool (p1,5.000000,15.500000,8.500000,\Rx:=0.000000,\Ry:=0.000000),vel1,zoneval,Extruder\WObj:=Workobject_1;
MoveL RelTool (p1,5.500000,15.500000,8.500000,\Rx:=0.000000,\Ry:=0.000000),vel1,zoneval,Extruder\WObj:=Workobject_1;
MoveL RelTool (p1,6.000000,15.500000,8.500000,\Rx:=0.000000,\Ry:=0.000000),vel1,zoneval,Extruder\WObj:=Workobject_1;
MoveL RelTool (p1,6.500000,15.500000,8.500000,\Rx:=0.000000,\Ry:=0.000000),vel1,zoneval,Extruder\WObj:=Workobject_1;
MoveL RelTool (p1,7.000000,15.500000,8.500000,\Rx:=0.000000,\Ry:=0.000000),vel1,zoneval,Extruder\WObj:=Workobject_1;
MoveL RelTool (p1,7.500000,15.500000,8.500000,\Rx:=0.000000,\Ry:=0.000000),vel1,zoneval,Extruder\WObj:=Workobject_1;
MoveL RelTool (p1,8.000000,15.500000,8.500000,\Rx:=0.000000,\Ry:=0.000000),vel1,zoneval,Extruder\WObj:=Workobject_1;
MoveL RelTool (p1,8.500000,15.500000,8.500000,\Rx:=0.000000,\Ry:=0.000000),vel1,zoneval,Extruder\WObj:=Workobject_1;
MoveL RelTool (p1,9.000000,15.500000,8.500000,\Rx:=0.000000,\Ry:=0.000000),vel1,zoneval,Extruder\WObj:=Workobject_1;
MoveL RelTool (p1,9.500000,15.500000,8.500000,\Rx:=0.000000,\Ry:=0.000000),vel1,zoneval,Extruder\WObj:=Workobject_1;
MoveL RelTool (p1,10.000000,15.500000,8.500000,\Rx:=0.000000,\Ry:=0.000000),vel1,zoneval,Extruder\WObj:=Workobject_1;
MoveL RelTool (p1,10.500000,15.500000,8.500000,\Rx:=0.000000,\Ry:=0.000000),vel1,zoneval,Extruder\WObj:=Workobject_1;
MoveL RelTool (p1,11.000000,15.500000,8.500000,\Rx:=0.000000,\Ry:=0.000000),vel1,zoneval,Extruder\WObj:=Workobject_1;
MoveL RelTool (p1,11.500000,15.500000,8.500000,\Rx:=0.000000,\Ry:=0.000000),vel1,zoneval,Extruder\WObj:=Workobject_1;
MoveL RelTool (p1,12.000000,15.500000,8.500000,\Rx:=0.000000,\Ry:=0.000000),vel1,zoneval,Extruder\WObj:=Workobject_1;
MoveL RelTool (p1,12.500000,15.500000,8.500000,\Rx:=0.000000,\Ry:=0.000000),vel1,zoneval,Extruder\WObj:=Workobject_1;
MoveL RelTool (p1,13.000000,15.500000,8.500000,\Rx:=0.000000,\Ry:=0.000000),vel1,zoneval,Extruder\WObj:=Workobject_1;
MoveL RelTool (p1,13.500000,15.500000,8.500000,\Rx:=0.000000,\Ry:=0.000000),vel1,zoneval,Extruder\WObj:=Workobject_1;
MoveL RelTool (p1,14.000000,15.500000,8.500000,\Rx:=0.000000,\Ry:=0.000000),vel1,zoneval,Extruder\WObj:=Workobject_1;
MoveL RelTool (p1,14.500000,15.500000,8.500000,\Rx:=0.000000,\Ry:=0.000000),vel1,zoneval,Extruder\WObj:=Workobject_1;
MoveL RelTool (p1,15.000000,15.500000,8.500000,\Rx:=0.000000,\Ry:=0.000000),vel1,zoneval,Extruder\WObj:=Workobject_1;
MoveL RelTool (p1,15.500000,15.500000,8.500000,\Rx:=0.000000,\Ry:=0.000000),vel1,zoneval,Extruder\WObj:=Workobject_1;
MoveL RelTool (p1,16.000000,15.500000,8.500000,\Rx:=0.000000,\Ry:=0.000000),vel1,zoneval,Extruder\WObj:=Workobject_1;
MoveL RelTool (p1,16.500000,15.500000,8.500000,\Rx:=0.000000,\Ry:=0.000000),vel1,zoneval,Extruder\WObj:=Workobject_1;
MoveL RelTool (p1,17.000000,15.500000,8.508911,\Rx:=0.000000,\Ry:=0.000000),vel1,zoneval,Extruder\WObj:=Workobject_1;
MoveL RelTool (p1,17.500000,15.500000,8.570628,\Rx:=0.000000,\Ry:=0.000000),vel1,zoneval,Extruder\WObj:=Workobject_1;
MoveL RelTool (p1,18.000000,15.500000,8.722633,\Rx:=0.000000,\Ry:=0.000000),vel1,zoneval,Extruder\WObj:=Workobject_1;
MoveL RelTool (p1,18.500000,15.500000,8.980296,\Rx:=0.000000,\Ry:=0.000000),vel1,zoneval,Extruder\WObj:=Workobject_1;
MoveL RelTool (p1,19.000000,15.500000,9.374813,\Rx:=0.000000,\Ry:=0.000000),vel1,zoneval,Extruder\WObj:=Workobject_1;
MoveL RelTool (p1,19.500000,15.500000,9.992651,\Rx:=0.000000,\Ry:=0.000000),vel1,zoneval,Extruder\WObj:=Workobject_1;
MoveL RelTool (p1,20.000000,15.500000,10.624391,\Rx:=0.000000,\Ry:=0.000000),vel1,zoneval,Extruder\WObj:=Workobject_1;
MoveL RelTool (p1,20.500000,15.500000,11.179913,\Rx:=0.000000,\Ry:=0.000000),vel1,zoneval,Extruder\WObj:=Workobject_1;
MoveL RelTool (p1,21.000000,15.500000,11.682592,\Rx:=0.000000,\Ry:=0.000000),vel1,zoneval,Extruder\WObj:=Workobject_1;
MoveL RelTool (p1,21.500000,15.500000,12.140557,\Rx:=0.000000,\Ry:=0.000000),vel1,zoneval,Extruder\WObj:=Workobject_1;
MoveL RelTool (p1,22.000000,15.500000,12.548016,\Rx:=0.000000,\Ry:=0.000000),vel1,zoneval,Extruder\WObj:=Workobject_1;
MoveL RelTool (p1,22.500000,15.500000,12.938538,\Rx:=0.000000,\Ry:=0.000000),vel1,zoneval,Extruder\WObj:=Workobject_1;
MoveL RelTool (p1,23.000000,15.500000,13.289470,\Rx:=0.000000,\Ry:=0.000000),vel1,zoneval,Extruder\WObj:=Workobject_1;
MoveL RelTool (p1,23.500000,15.500000,13.627415,\Rx:=0.000000,\Ry:=0.000000),vel1,zoneval,Extruder\WObj:=Workobject_1;
MoveL RelTool (p1,24.000000,15.500000,13.936113,\Rx:=0.000000,\Ry:=0.000000),vel1,zoneval,Extruder\WObj:=Workobject_1;
MoveL RelTool (p1,24.500000,15.500000,14.234470,\Rx:=0.000000,\Ry:=0.000000),vel1,zoneval,Extruder\WObj:=Workobject_1;
MoveL RelTool (p1,25.000000,15.500000,14.505671,\Rx:=0.000000,\Ry:=0.000000),vel1,zoneval,Extruder\WObj:=Workobject_1;
MoveL RelTool (p1,25.500000,15.500000,14.776617,\Rx:=0.000000,\Ry:=0.000000),vel1,zoneval,Extruder\WObj:=Workobject_1;
MoveL RelTool (p1,26.000000,15.500000,15.015915,\Rx:=0.000000,\Ry:=0.000000),vel1,zoneval,Extruder\WObj:=Workobject_1;
MoveL RelTool (p1,26.500000,15.500000,15.253666,\Rx:=0.000000,\Ry:=0.000000),vel1,zoneval,Extruder\WObj:=Workobject_1;
MoveL RelTool (p1,27.000000,15.500000,15.474790,\Rx:=0.000000,\Ry:=0.000000),vel1,zoneval,Extruder\WObj:=Workobject_1;
MoveL RelTool (p1,27.500000,15.500000,15.682626,\Rx:=0.000000,\Ry:=0.000000),vel1,zoneval,Extruder\WObj:=Workobject_1;
MoveL RelTool (p1,28.000000,15.500000,15.890462,\Rx:=0.000000,\Ry:=0.000000),vel1,zoneval,Extruder\WObj:=Workobject_1;
MoveL RelTool (p1,28.500000,15.500000,16.075120,\Rx:=0.000000,\Ry:=0.000000),vel1,zoneval,Extruder\WObj:=Workobject_1;
MoveL RelTool (p1,29.000000,15.500000,16.256120,\Rx:=0.000000,\Ry:=0.000000),vel1,zoneval,Extruder\WObj:=Workobject_1;
MoveL RelTool (p1,29.500000,15.500000,16.435168,\Rx:=0.000000,\Ry:=0.000000),vel1,zoneval,Extruder\WObj:=Workobject_1;
MoveL RelTool (p1,30.000000,15.500000,16.591832,\Rx:=0.000000,\Ry:=0.000000),vel1,zoneval,Extruder\WObj:=Workobject_1;
MoveL RelTool (p1,30.500000,15.500000,16.747901,\Rx:=0.000000,\Ry:=0.000000),vel1,zoneval,Extruder\WObj:=Workobject_1;
MoveL RelTool (p1,31.000000,15.500000,16.901822,\Rx:=0.000000,\Ry:=0.000000),vel1,zoneval,Extruder\WObj:=Workobject_1;
MoveL RelTool (p1,31.500000,15.500000,17.034226,\Rx:=0.000000,\Ry:=0.000000),vel1,zoneval,Extruder\WObj:=Workobject_1;
MoveL RelTool (p1,32.000000,15.500000,17.166631,\Rx:=0.000000,\Ry:=0.000000),vel1,zoneval,Extruder\WObj:=Workobject_1;
MoveL RelTool (p1,32.500000,15.500000,17.298270,\Rx:=0.000000,\Ry:=0.000000),vel1,zoneval,Extruder\WObj:=Workobject_1;
MoveL RelTool (p1,33.000000,15.500000,17.409691,\Rx:=0.000000,\Ry:=0.000000),vel1,zoneval,Extruder\WObj:=Workobject_1;
MoveL RelTool (p1,33.500000,15.500000,17.519618,\Rx:=0.000000,\Ry:=0.000000),vel1,zoneval,Extruder\WObj:=Workobject_1;
MoveL RelTool (p1,34.000000,15.500000,17.629544,\Rx:=0.000000,\Ry:=0.000000),vel1,zoneval,Extruder\WObj:=Workobject_1;
MoveL RelTool (p1,34.500000,15.500000,17.722158,\Rx:=0.000000,\Ry:=0.000000),vel1,zoneval,Extruder\WObj:=Workobject_1;
MoveL RelTool (p1,35.000000,15.500000,17.810731,\Rx:=0.000000,\Ry:=0.000000),vel1,zoneval,Extruder\WObj:=Workobject_1;
MoveL RelTool (p1,35.500000,15.500000,17.899305,\Rx:=0.000000,\Ry:=0.000000),vel1,zoneval,Extruder\WObj:=Workobject_1;
MoveL RelTool (p1,36.000000,15.500000,17.980675,\Rx:=0.000000,\Ry:=0.000000),vel1,zoneval,Extruder\WObj:=Workobject_1;
MoveL RelTool (p1,36.500000,15.500000,18.048938,\Rx:=0.000000,\Ry:=0.000000),vel1,zoneval,Extruder\WObj:=Workobject_1;
MoveL RelTool (p1,37.000000,15.500000,18.117203,\Rx:=0.000000,\Ry:=0.000000),vel1,zoneval,Extruder\WObj:=Workobject_1;
MoveL RelTool (p1,37.500000,15.500000,18.184708,\Rx:=0.000000,\Ry:=0.000000),vel1,zoneval,Extruder\WObj:=Workobject_1;
MoveL RelTool (p1,38.000000,15.500000,18.233311,\Rx:=0.000000,\Ry:=0.000000),vel1,zoneval,Extruder\WObj:=Workobject_1;
MoveL RelTool (p1,38.500000,15.500000,18.281914,\Rx:=0.000000,\Ry:=0.000000),vel1,zoneval,Extruder\WObj:=Workobject_1;
MoveL RelTool (p1,39.000000,15.500000,18.330517,\Rx:=0.000000,\Ry:=0.000000),vel1,zoneval,Extruder\WObj:=Workobject_1;
MoveL RelTool (p1,39.500000,15.500000,18.371829,\Rx:=0.000000,\Ry:=0.000000),vel1,zoneval,Extruder\WObj:=Workobject_1;
MoveL RelTool (p1,40.000000,15.500000,18.401279,\Rx:=0.000000,\Ry:=0.000000),vel1,zoneval,Extruder\WObj:=Workobject_1;
MoveL RelTool (p1,40.500000,15.500000,18.430729,\Rx:=0.000000,\Ry:=0.000000),vel1,zoneval,Extruder\WObj:=Workobject_1;
MoveL RelTool (p1,41.000000,15.500000,18.459969,\Rx:=0.000000,\Ry:=0.000000),vel1,zoneval,Extruder\WObj:=Workobject_1;
MoveL RelTool (p1,41.500000,15.500000,18.472422,\Rx:=0.000000,\Ry:=0.000000),vel1,zoneval,Extruder\WObj:=Workobject_1;
MoveL RelTool (p1,42.000000,15.500000,18.482833,\Rx:=0.000000,\Ry:=0.000000),vel1,zoneval,Extruder\WObj:=Workobject_1;
MoveL RelTool (p1,42.500000,15.500000,18.493245,\Rx:=0.000000,\Ry:=0.000000),vel1,zoneval,Extruder\WObj:=Workobject_1;
MoveL RelTool (p1,43.000000,15.500000,18.497115,\Rx:=0.000000,\Ry:=0.000000),vel1,zoneval,Extruder\WObj:=Workobject_1;
MoveL RelTool (p1,43.500000,15.500000,18.488586,\Rx:=0.000000,\Ry:=0.000000),vel1,zoneval,Extruder\WObj:=Workobject_1;
MoveL RelTool (p1,44.000000,15.500000,18.480057,\Rx:=0.000000,\Ry:=0.000000),vel1,zoneval,Extruder\WObj:=Workobject_1;
MoveL RelTool (p1,44.500000,15.500000,18.471528,\Rx:=0.000000,\Ry:=0.000000),vel1,zoneval,Extruder\WObj:=Workobject_1;
MoveL RelTool (p1,45.000000,15.500000,18.448105,\Rx:=0.000000,\Ry:=0.000000),vel1,zoneval,Extruder\WObj:=Workobject_1;
MoveL RelTool (p1,45.500000,15.500000,18.420561,\Rx:=0.000000,\Ry:=0.000000),vel1,zoneval,Extruder\WObj:=Workobject_1;
MoveL RelTool (p1,46.000000,15.500000,18.393017,\Rx:=0.000000,\Ry:=0.000000),vel1,zoneval,Extruder\WObj:=Workobject_1;
MoveL RelTool (p1,46.500000,15.500000,18.360568,\Rx:=0.000000,\Ry:=0.000000),vel1,zoneval,Extruder\WObj:=Workobject_1;
MoveL RelTool (p1,47.000000,15.500000,18.313937,\Rx:=0.000000,\Ry:=0.000000),vel1,zoneval,Extruder\WObj:=Workobject_1;
MoveL RelTool (p1,47.500000,15.500000,18.267305,\Rx:=0.000000,\Ry:=0.000000),vel1,zoneval,Extruder\WObj:=Workobject_1;
MoveL RelTool (p1,48.000000,15.500000,18.220674,\Rx:=0.000000,\Ry:=0.000000),vel1,zoneval,Extruder\WObj:=Workobject_1;
MoveL RelTool (p1,48.500000,15.500000,18.160235,\Rx:=0.000000,\Ry:=0.000000),vel1,zoneval,Extruder\WObj:=Workobject_1;
MoveL RelTool (p1,49.000000,15.500000,18.094178,\Rx:=0.000000,\Ry:=0.000000),vel1,zoneval,Extruder\WObj:=Workobject_1;
MoveL RelTool (p1,49.500000,15.500000,18.028121,\Rx:=0.000000,\Ry:=0.000000),vel1,zoneval,Extruder\WObj:=Workobject_1;
MoveL RelTool (p1,50.000000,15.500000,17.954415,\Rx:=0.000000,\Ry:=0.000000),vel1,zoneval,Extruder\WObj:=Workobject_1;
MoveL RelTool (p1,50.500000,15.500000,17.868439,\Rx:=0.000000,\Ry:=0.000000),vel1,zoneval,Extruder\WObj:=Workobject_1;
MoveL RelTool (p1,51.000000,15.500000,17.782462,\Rx:=0.000000,\Ry:=0.000000),vel1,zoneval,Extruder\WObj:=Workobject_1;
MoveL RelTool (p1,51.500000,15.500000,17.696850,\Rx:=0.000000,\Ry:=0.000000),vel1,zoneval,Extruder\WObj:=Workobject_1;
MoveL RelTool (p1,52.000000,15.500000,17.590416,\Rx:=0.000000,\Ry:=0.000000),vel1,zoneval,Extruder\WObj:=Workobject_1;
MoveL RelTool (p1,52.500000,15.500000,17.483661,\Rx:=0.000000,\Ry:=0.000000),vel1,zoneval,Extruder\WObj:=Workobject_1;
MoveL RelTool (p1,53.000000,15.500000,17.376906,\Rx:=0.000000,\Ry:=0.000000),vel1,zoneval,Extruder\WObj:=Workobject_1;
MoveL RelTool (p1,53.500000,15.500000,17.249829,\Rx:=0.000000,\Ry:=0.000000),vel1,zoneval,Extruder\WObj:=Workobject_1;
MoveL RelTool (p1,54.000000,15.500000,17.121229,\Rx:=0.000000,\Ry:=0.000000),vel1,zoneval,Extruder\WObj:=Workobject_1;
MoveL RelTool (p1,54.500000,15.500000,16.992629,\Rx:=0.000000,\Ry:=0.000000),vel1,zoneval,Extruder\WObj:=Workobject_1;
MoveL RelTool (p1,55.000000,15.500000,16.847593,\Rx:=0.000000,\Ry:=0.000000),vel1,zoneval,Extruder\WObj:=Workobject_1;
MoveL RelTool (p1,55.500000,15.500000,16.695978,\Rx:=0.000000,\Ry:=0.000000),vel1,zoneval,Extruder\WObj:=Workobject_1;
MoveL RelTool (p1,56.000000,15.500000,16.544363,\Rx:=0.000000,\Ry:=0.000000),vel1,zoneval,Extruder\WObj:=Workobject_1;
MoveL RelTool (p1,56.500000,15.500000,16.372394,\Rx:=0.000000,\Ry:=0.000000),vel1,zoneval,Extruder\WObj:=Workobject_1;
MoveL RelTool (p1,57.000000,15.500000,16.196484,\Rx:=0.000000,\Ry:=0.000000),vel1,zoneval,Extruder\WObj:=Workobject_1;
MoveL RelTool (p1,57.500000,15.500000,16.019130,\Rx:=0.000000,\Ry:=0.000000),vel1,zoneval,Extruder\WObj:=Workobject_1;
MoveL RelTool (p1,58.000000,15.500000,15.817503,\Rx:=0.000000,\Ry:=0.000000),vel1,zoneval,Extruder\WObj:=Workobject_1;
MoveL RelTool (p1,58.500000,15.500000,15.615877,\Rx:=0.000000,\Ry:=0.000000),vel1,zoneval,Extruder\WObj:=Workobject_1;
MoveL RelTool (p1,59.000000,15.500000,15.403433,\Rx:=0.000000,\Ry:=0.000000),vel1,zoneval,Extruder\WObj:=Workobject_1;
MoveL RelTool (p1,59.500000,15.500000,15.173636,\Rx:=0.000000,\Ry:=0.000000),vel1,zoneval,Extruder\WObj:=Workobject_1;
MoveL RelTool (p1,60.000000,15.500000,14.942281,\Rx:=0.000000,\Ry:=0.000000),vel1,zoneval,Extruder\WObj:=Workobject_1;
MoveL RelTool (p1,60.500000,15.500000,14.681236,\Rx:=0.000000,\Ry:=0.000000),vel1,zoneval,Extruder\WObj:=Workobject_1;
MoveL RelTool (p1,61.000000,15.500000,14.420190,\Rx:=0.000000,\Ry:=0.000000),vel1,zoneval,Extruder\WObj:=Workobject_1;
MoveL RelTool (p1,61.500000,15.500000,14.133931,\Rx:=0.000000,\Ry:=0.000000),vel1,zoneval,Extruder\WObj:=Workobject_1;
MoveL RelTool (p1,62.000000,15.500000,13.837956,\Rx:=0.000000,\Ry:=0.000000),vel1,zoneval,Extruder\WObj:=Workobject_1;
MoveL RelTool (p1,62.500000,15.500000,13.514260,\Rx:=0.000000,\Ry:=0.000000),vel1,zoneval,Extruder\WObj:=Workobject_1;
MoveL RelTool (p1,63.000000,15.500000,13.178888,\Rx:=0.000000,\Ry:=0.000000),vel1,zoneval,Extruder\WObj:=Workobject_1;
MoveL RelTool (p1,63.500000,15.500000,12.806751,\Rx:=0.000000,\Ry:=0.000000),vel1,zoneval,Extruder\WObj:=Workobject_1;
MoveL RelTool (p1,64.000000,15.500000,12.421133,\Rx:=0.000000,\Ry:=0.000000),vel1,zoneval,Extruder\WObj:=Workobject_1;
MoveL RelTool (p1,64.500000,15.500000,11.988319,\Rx:=0.000000,\Ry:=0.000000),vel1,zoneval,Extruder\WObj:=Workobject_1;
MoveL RelTool (p1,65.000000,15.500000,11.517461,\Rx:=0.000000,\Ry:=0.000000),vel1,zoneval,Extruder\WObj:=Workobject_1;
MoveL RelTool (p1,65.500000,15.500000,11.005999,\Rx:=0.000000,\Ry:=0.000000),vel1,zoneval,Extruder\WObj:=Workobject_1;
MoveL RelTool (p1,66.000000,15.500000,10.428127,\Rx:=0.000000,\Ry:=0.000000),vel1,zoneval,Extruder\WObj:=Workobject_1;
MoveL RelTool (p1,66.500000,15.500000,9.763981,\Rx:=0.000000,\Ry:=0.000000),vel1,zoneval,Extruder\WObj:=Workobject_1;
MoveL RelTool (p1,67.000000,15.500000,9.225973,\Rx:=0.000000,\Ry:=0.000000),vel1,zoneval,Extruder\WObj:=Workobject_1;
MoveL RelTool (p1,67.500000,15.500000,8.874086,\Rx:=0.000000,\Ry:=0.000000),vel1,zoneval,Extruder\WObj:=Workobject_1;
MoveL RelTool (p1,68.000000,15.500000,8.652682,\Rx:=0.000000,\Ry:=0.000000),vel1,zoneval,Extruder\WObj:=Workobject_1;
MoveL RelTool (p1,68.500000,15.500000,8.535785,\Rx:=0.000000,\Ry:=0.000000),vel1,zoneval,Extruder\WObj:=Workobject_1;
MoveL RelTool (p1,69.000000,15.500000,8.500000,\Rx:=0.000000,\Ry:=0.000000),vel1,zoneval,Extruder\WObj:=Workobject_1;
MoveL RelTool (p1,69.500000,15.500000,8.500000,\Rx:=0.000000,\Ry:=0.000000),vel1,zoneval,Extruder\WObj:=Workobject_1;
MoveL RelTool (p1,70.000000,15.500000,8.500000,\Rx:=0.000000,\Ry:=0.000000),vel1,zoneval,Extruder\WObj:=Workobject_1;
MoveL RelTool (p1,70.500000,15.500000,8.500000,\Rx:=0.000000,\Ry:=0.000000),vel1,zoneval,Extruder\WObj:=Workobject_1;
MoveL RelTool (p1,71.000000,15.500000,8.500000,\Rx:=0.000000,\Ry:=0.000000),vel1,zoneval,Extruder\WObj:=Workobject_1;
MoveL RelTool (p1,71.500000,15.500000,8.500000,\Rx:=0.000000,\Ry:=0.000000),vel1,zoneval,Extruder\WObj:=Workobject_1;
MoveL RelTool (p1,72.000000,15.500000,8.500000,\Rx:=0.000000,\Ry:=0.000000),vel1,zoneval,Extruder\WObj:=Workobject_1;
MoveL RelTool (p1,72.500000,15.500000,8.500000,\Rx:=0.000000,\Ry:=0.000000),vel1,zoneval,Extruder\WObj:=Workobject_1;
MoveL RelTool (p1,73.000000,15.500000,8.500000,\Rx:=0.000000,\Ry:=0.000000),vel1,zoneval,Extruder\WObj:=Workobject_1;
MoveL RelTool (p1,73.500000,15.500000,8.500000,\Rx:=0.000000,\Ry:=0.000000),vel1,zoneval,Extruder\WObj:=Workobject_1;
MoveL RelTool (p1,74.000000,15.500000,8.500000,\Rx:=0.000000,\Ry:=0.000000),vel1,zoneval,Extruder\WObj:=Workobject_1;
MoveL RelTool (p1,74.500000,15.500000,8.500000,\Rx:=0.000000,\Ry:=0.000000),vel1,zoneval,Extruder\WObj:=Workobject_1;
MoveL RelTool (p1,75.000000,15.500000,8.500000,\Rx:=0.000000,\Ry:=0.000000),vel1,zoneval,Extruder\WObj:=Workobject_1;
MoveL RelTool (p1,75.500000,15.500000,8.500000,\Rx:=0.000000,\Ry:=0.000000),vel1,zoneval,Extruder\WObj:=Workobject_1;
MoveL RelTool (p1,76.000000,15.500000,8.500000,\Rx:=0.000000,\Ry:=0.000000),vel1,zoneval,Extruder\WObj:=Workobject_1;
MoveL RelTool (p1,76.500000,15.500000,8.500000,\Rx:=0.000000,\Ry:=0.000000),vel1,zoneval,Extruder\WObj:=Workobject_1;
MoveL RelTool (p1,77.000000,15.500000,8.500000,\Rx:=0.000000,\Ry:=0.000000),vel1,zoneval,Extruder\WObj:=Workobject_1;
MoveL RelTool (p1,77.500000,15.500000,8.500000,\Rx:=0.000000,\Ry:=0.000000),vel1,zoneval,Extruder\WObj:=Workobject_1;
MoveL RelTool (p1,78.000000,15.500000,8.500000,\Rx:=0.000000,\Ry:=0.000000),vel1,zoneval,Extruder\WObj:=Workobject_1;
MoveL RelTool (p1,78.500000,15.500000,8.500000,\Rx:=0.000000,\Ry:=0.000000),vel1,zoneval,Extruder\WObj:=Workobject_1;
MoveL RelTool (p1,79.000000,15.500000,8.500000,\Rx:=0.000000,\Ry:=0.000000),vel1,zoneval,Extruder\WObj:=Workobject_1;
MoveL RelTool (p1,79.500000,15.500000,8.500000,\Rx:=0.000000,\Ry:=0.000000),vel1,zoneval,Extruder\WObj:=Workobject_1;
MoveL RelTool (p1,80.000000,15.500000,8.500000,\Rx:=0.000000,\Ry:=0.000000),vel1,zoneval,Extruder\WObj:=Workobject_1;
MoveL RelTool (p1,80.500000,15.500000,8.500000,\Rx:=0.000000,\Ry:=0.000000),vel1,zoneval,Extruder\WObj:=Workobject_1;
MoveL RelTool (p1,81.000000,15.500000,8.500000,\Rx:=0.000000,\Ry:=0.000000),vel1,zoneval,Extruder\WObj:=Workobject_1;
MoveL RelTool (p1,81.500000,15.500000,8.500000,\Rx:=0.000000,\Ry:=0.000000),vel1,zoneval,Extruder\WObj:=Workobject_1;
MoveL RelTool (p1,82.000000,15.500000,8.500000,\Rx:=0.000000,\Ry:=0.000000),vel1,zoneval,Extruder\WObj:=Workobject_1;
SetDO Test_Out, 1;
MoveL RelTool (p1,82.000000,15.500000,70.00000,\Rx:=0.000000,\Ry:=0.000000),vel1,zoneval,Extruder\WObj:=Workobject_1;

MoveL RelTool (p1,3.000000,3.000000,70.000000,\Rx:=0.000000,\Ry:=0.000000),vel1,z0,Extruder\WObj:=Workobject_1;
MoveL RelTool (p1,3.000000,3.000000,9.000000,\Rx:=0.000000,\Ry:=0.000000),vel1,z0,Extruder\WObj:=Workobject_1;
SetDO Test_Out, 0;
WaitTime 2;

